C05474=1205.016,78.831,-47.924,-178.902,5.757,148.692
C05475=1205.020,78.581,-47.907,-178.904,5.757,148.692
C05476=1205.025,78.332,-47.889,-178.907,5.756,148.693
C05477=1205.030,78.082,-47.872,-178.910,5.754,148.693
C05478=1205.035,77.833,-47.854,-178.912,5.754,148.694
C05479=1205.039,77.584,-47.836,-178.915,5.753,148.695
C05480=1205.044,77.335,-47.819,-178.917,5.752,148.695
C05481=1205.049,77.085,-47.801,-178.920,5.752,148.696
C05482=1205.055,76.836,-47.784,-178.922,5.750,148.696
C05483=1205.059,76.587,-47.766,-178.925,5.749,148.697
C05484=1205.064,76.337,-47.749,-178.928,5.749,148.698
C05485=1205.069,76.088,-47.731,-178.930,5.748,148.698
C05486=1205.073,75.838,-47.714,-178.933,5.747,148.699
C05487=1205.079,75.590,-47.697,-178.936,5.746,148.699
C05488=1205.084,75.340,-47.680,-178.938,5.745,148.700
C05489=1205.089,75.091,-47.662,-178.940,5.745,148.700
C05490=1205.093,74.841,-47.645,-178.943,5.744,148.701
C05491=1205.099,74.592,-47.628,-178.946,5.742,148.701
C05492=1205.104,74.342,-47.610,-178.948,5.742,148.702
C05493=1205.108,74.093,-47.593,-178.951,5.741,148.703
C05494=1205.113,73.844,-47.575,-178.953,5.740,148.703
C05495=1205.117,73.594,-47.558,-178.956,5.740,148.704
C05496=1205.122,73.345,-47.540,-178.959,5.738,148.704
C05497=1205.128,73.096,-47.523,-178.961,5.737,148.705
C05498=1205.133,72.846,-47.507,-178.964,5.737,148.706
C05499=1205.138,72.597,-47.489,-178.966,5.736,148.706
C05500=1205.143,72.348,-47.472,-178.968,5.735,148.707
C05501=1205.147,72.098,-47.455,-178.972,5.734,148.707
C05502=1205.152,71.849,-47.437,-178.974,5.733,148.708
C05503=1205.157,71.599,-47.420,-178.976,5.732,148.708
C05504=1205.163,71.350,-47.403,-178.979,5.732,148.709
C05505=1205.167,71.101,-47.385,-178.982,5.731,148.710
C05506=1205.172,70.852,-47.369,-178.984,5.730,148.710
C05507=1205.177,70.602,-47.351,-178.987,5.729,148.711
C05508=1205.181,70.353,-47.334,-178.990,5.729,148.711
C05509=1205.187,70.103,-47.317,-178.992,5.728,148.712
C05510=1205.192,69.854,-47.300,-178.994,5.727,148.713
C05511=1205.197,69.605,-47.283,-178.998,5.726,148.713
C05512=1205.201,69.356,-47.266,-179.000,5.725,148.714
C05513=1205.206,69.106,-47.249,-179.002,5.724,148.714
C05514=1205.211,68.856,-47.231,-179.005,5.724,148.715
C05515=1205.216,68.607,-47.215,-179.007,5.723,148.715
C05516=1205.221,68.358,-47.197,-179.010,5.722,148.716
C05517=1205.226,68.109,-47.180,-179.013,5.721,148.717
C05518=1205.231,67.859,-47.163,-179.015,5.720,148.717
C05519=1205.236,67.609,-47.146,-179.018,5.719,148.718
C05520=1205.241,67.360,-47.130,-179.020,5.719,148.718
C05521=1205.246,67.111,-47.112,-179.023,5.718,148.719
C05522=1205.250,66.862,-47.095,-179.026,5.716,148.720
C05523=1205.255,66.612,-47.078,-179.028,5.716,148.720
C05524=1205.260,66.363,-47.062,-179.031,5.715,148.721
C05525=1205.266,66.114,-47.045,-179.033,5.714,148.721
C05526=1205.270,65.864,-47.028,-179.036,5.714,148.722
C05527=1205.275,65.614,-47.011,-179.038,5.713,148.723
C05528=1205.280,65.365,-46.994,-179.041,5.712,148.723
C05529=1205.285,65.116,-46.976,-179.044,5.711,148.724
C05530=1205.290,64.867,-46.960,-179.046,5.711,148.724
C05531=1205.294,64.617,-46.943,-179.049,5.710,148.725
C05532=1205.299,64.368,-46.926,-179.051,5.709,148.726
C05533=1205.305,64.119,-46.910,-179.054,5.709,148.726
C05534=1205.310,63.869,-46.892,-179.056,5.708,148.727
C05535=1205.314,63.620,-46.876,-179.059,5.706,148.727
C05536=1205.319,63.370,-46.859,-179.062,5.706,148.728
C05537=1205.325,63.121,-46.842,-179.064,5.705,148.729
C05538=1205.329,62.871,-46.825,-179.067,5.704,148.729
C05539=1205.334,62.622,-46.808,-179.069,5.704,148.730
C05540=1205.339,62.373,-46.792,-179.072,5.703,148.730
C05541=1205.344,62.123,-46.775,-179.074,5.702,148.731
C05542=1205.349,61.874,-46.758,-179.077,5.701,148.731
C05543=1205.354,61.625,-46.742,-179.080,5.700,148.732
C05544=1205.359,61.375,-46.725,-179.082,5.700,148.733
C05545=1205.364,61.126,-46.708,-179.085,5.699,148.733
C05546=1205.368,60.876,-46.691,-179.087,5.698,148.734
C05547=1205.373,60.627,-46.675,-179.090,5.698,148.735
C05548=1205.379,60.377,-46.657,-179.092,5.697,148.735
C05549=1205.383,60.128,-46.641,-179.095,5.695,148.736
C05550=1205.388,59.879,-46.624,-179.098,5.695,148.736
C05551=1205.393,59.629,-46.607,-179.100,5.694,148.737
C05552=1205.398,59.380,-46.590,-179.103,5.693,148.737
C05553=1205.403,59.131,-46.575,-179.105,5.693,148.738
C05554=1205.408,58.881,-46.558,-179.108,5.692,148.739
C05555=1205.414,58.632,-46.541,-179.110,5.691,148.739
C05556=1205.418,58.382,-46.525,-179.113,5.691,148.740
C05557=1205.422,58.133,-46.508,-179.116,5.690,148.741
C05558=1205.428,57.884,-46.492,-179.118,5.689,148.741
C05559=1205.433,57.634,-46.474,-179.121,5.688,148.742
C05560=1205.438,57.384,-46.458,-179.123,5.688,148.742
C05561=1205.443,57.136,-46.442,-179.126,5.687,148.743
C05562=1205.447,56.886,-46.425,-179.128,5.686,148.743
C05563=1205.453,56.637,-46.409,-179.131,5.686,148.744
C05564=1205.457,56.387,-46.392,-179.133,5.685,148.745
C05565=1205.462,56.137,-46.376,-179.137,5.684,148.745
C05566=1205.467,55.889,-46.360,-179.139,5.683,148.746
C05567=1205.473,55.639,-46.342,-179.141,5.682,148.746
C05568=1205.478,55.371,-46.325,-179.144,5.682,148.747
C05569=1205.483,55.102,-46.307,-179.147,5.681,148.748
C05570=1205.488,54.834,-46.290,-179.150,5.680,148.748
C05571=1205.494,54.565,-46.272,-179.152,5.679,148.749
C05572=1205.499,54.316,-46.255,-179.155,5.679,148.750
C05573=1205.503,54.066,-46.239,-179.157,5.678,148.750
C05574=1205.509,53.817,-46.223,-179.160,5.677,148.751
C05575=1205.513,53.567,-46.206,-179.162,5.677,148.752
C05576=1205.518,53.318,-46.190,-179.165,5.676,148.752
C05577=1205.523,53.068,-46.174,-179.167,5.675,148.753
C05578=1205.529,52.819,-46.157,-179.170,5.674,148.753
C05579=1205.533,52.570,-46.141,-179.173,5.673,148.754
C05580=1205.539,52.320,-46.125,-179.175,5.672,148.754
C05581=1205.543,52.071,-46.108,-179.178,5.672,148.755
C05582=1205.548,51.821,-46.092,-179.181,5.671,148.756
C05583=1205.553,51.572,-46.076,-179.183,5.671,148.756
C05584=1205.557,51.323,-46.059,-179.185,5.670,148.757
C05585=1205.563,51.073,-46.044,-179.188,5.669,148.758
C05586=1205.567,50.824,-46.027,-179.191,5.669,148.758
C05587=1205.572,50.575,-46.011,-179.193,5.668,148.759
C05588=1205.577,50.325,-45.995,-179.195,5.667,148.759
C05589=1205.583,50.076,-45.978,-179.198,5.667,148.760
C05590=1205.588,49.826,-45.962,-179.201,5.665,148.761
C05591=1205.593,49.577,-45.946,-179.204,5.665,148.761
C05592=1205.597,49.327,-45.929,-179.206,5.664,148.762
C05593=1205.603,49.078,-45.913,-179.209,5.663,148.762
C05594=1205.607,48.828,-45.897,-179.211,5.663,148.763
C05595=1205.613,48.579,-45.881,-179.214,5.662,148.764
C05596=1205.617,48.329,-45.864,-179.216,5.661,148.764
C05597=1205.622,48.080,-45.849,-179.219,5.661,148.765
C05598=1205.627,47.831,-45.832,-179.221,5.660,148.766
C05599=1205.632,47.581,-45.817,-179.224,5.660,148.766
C05600=1205.637,47.332,-45.800,-179.226,5.659,148.767
C05601=1205.642,47.082,-45.784,-179.229,5.658,148.767
C05602=1205.647,46.834,-45.768,-179.231,5.658,148.768
C05603=1205.652,46.583,-45.752,-179.234,5.657,148.769
C05604=1205.657,46.334,-45.737,-179.237,5.656,148.769
C05605=1205.662,46.085,-45.720,-179.239,5.655,148.770
C05606=1205.667,45.835,-45.704,-179.242,5.654,148.770
C05607=1205.672,45.586,-45.688,-179.245,5.654,148.771
C05608=1205.677,45.336,-45.672,-179.247,5.653,148.772
C05609=1205.682,45.087,-45.655,-179.249,5.653,148.772
C05610=1205.686,44.838,-45.640,-179.252,5.652,148.773
C05611=1205.692,44.588,-45.625,-179.255,5.651,148.774
C05612=1205.696,44.339,-45.608,-179.257,5.651,148.774
C05613=1205.702,44.089,-45.593,-179.260,5.650,148.775
C05614=1205.706,43.839,-45.577,-179.262,5.649,148.775
C05615=1205.711,43.591,-45.560,-179.265,5.649,148.776
C05616=1205.717,43.341,-45.545,-179.267,5.648,148.777
C05617=1205.722,43.091,-45.529,-179.270,5.648,148.777
C05618=1205.727,42.842,-45.512,-179.272,5.647,148.778
C05619=1205.731,42.592,-45.496,-179.275,5.646,148.779
C05620=1205.737,42.343,-45.481,-179.278,5.646,148.779
C05621=1205.741,42.094,-45.465,-179.280,5.645,148.780
C05622=1205.746,41.844,-45.449,-179.282,5.644,148.780
C05623=1205.751,41.595,-45.434,-179.285,5.644,148.781
C05624=1205.756,41.345,-45.418,-179.288,5.643,148.782
C05625=1205.761,41.096,-45.401,-179.291,5.642,148.782
C05626=1205.767,40.846,-45.386,-179.293,5.641,148.783
C05627=1205.771,40.596,-45.370,-179.296,5.641,148.783
C05628=1205.776,40.347,-45.355,-179.298,5.640,148.784
C05629=1205.781,40.098,-45.339,-179.301,5.640,148.785
C05630=1205.786,39.848,-45.323,-179.304,5.639,148.785
C05631=1205.791,39.599,-45.307,-179.306,5.638,148.786
C05632=1205.797,39.350,-45.291,-179.308,5.638,148.787
C05633=1205.800,39.100,-45.275,-179.311,5.637,148.787
C05634=1205.806,38.851,-45.260,-179.314,5.637,148.788
C05635=1205.811,38.602,-45.244,-179.316,5.636,148.788
C05636=1205.816,38.351,-45.228,-179.318,5.635,148.789
C05637=1205.821,38.102,-45.213,-179.321,5.635,148.790
C05638=1205.826,37.853,-45.198,-179.324,5.634,148.790
C05639=1205.831,37.604,-45.181,-179.326,5.634,148.791
C05640=1205.836,37.354,-45.165,-179.328,5.633,148.792
C05641=1205.841,37.105,-45.150,-179.331,5.632,148.792
C05642=1205.845,36.855,-45.134,-179.334,5.632,148.793
C05643=1205.851,36.606,-45.119,-179.336,5.631,148.794
C05644=1205.856,36.356,-45.103,-179.339,5.630,148.794
C05645=1205.862,36.107,-45.088,-179.341,5.630,148.795
C05646=1205.866,35.857,-45.072,-179.344,5.629,148.795
C05647=1205.871,35.608,-45.057,-179.347,5.629,148.796
C05648=1205.876,35.358,-45.041,-179.349,5.628,148.797
C05649=1205.881,35.109,-45.024,-179.352,5.627,148.797
C05650=1205.885,34.860,-45.009,-179.354,5.627,148.798
C05651=1205.891,34.610,-44.994,-179.357,5.626,148.799
C05652=1205.896,34.361,-44.978,-179.359,5.626,148.799
C05653=1205.900,34.111,-44.963,-179.362,5.625,148.800
C05654=1205.906,33.862,-44.947,-179.365,5.624,148.801
C05655=1205.911,33.612,-44.932,-179.367,5.624,148.801
C05656=1205.916,33.363,-44.917,-179.369,5.623,148.802
C05657=1205.921,33.113,-44.901,-179.372,5.623,148.802
C05658=1205.926,32.864,-44.885,-179.375,5.622,148.803
C05659=1205.931,32.614,-44.870,-179.377,5.621,148.804
C05660=1205.936,32.365,-44.855,-179.379,5.621,148.804
C05661=1205.941,32.115,-44.839,-179.382,5.620,148.805
C05662=1205.945,31.866,-44.824,-179.385,5.620,148.805
C05663=1205.951,31.616,-44.808,-179.387,5.619,148.806
C05664=1205.956,31.367,-44.794,-179.390,5.618,148.807
C05665=1205.961,31.117,-44.778,-179.392,5.618,148.807
C05666=1205.966,30.867,-44.762,-179.395,5.617,148.808
C05667=1205.971,30.618,-44.747,-179.397,5.617,148.809
C05668=1205.976,30.369,-44.732,-179.400,5.616,148.809
C05669=1205.981,30.120,-44.717,-179.403,5.615,148.810
C05670=1205.986,29.870,-44.701,-179.405,5.615,148.810
C05671=1205.991,29.620,-44.685,-179.407,5.614,148.811
C05672=1205.996,29.351,-44.669,-179.410,5.614,148.812
C05673=1206.001,29.083,-44.652,-179.413,5.613,148.812
C05674=1206.007,28.814,-44.637,-179.415,5.613,148.813
C05675=1206.012,28.546,-44.620,-179.418,5.612,148.814
C05676=1206.017,28.296,-44.604,-179.421,5.611,148.815
C05677=1206.022,28.046,-44.590,-179.423,5.611,148.815
C05678=1206.028,27.797,-44.574,-179.426,5.610,148.816
C05679=1206.032,27.548,-44.559,-179.429,5.610,148.817
C05680=1206.037,27.298,-44.543,-179.431,5.609,148.817
C05681=1206.042,27.049,-44.528,-179.433,5.608,148.818
C05682=1206.048,26.799,-44.513,-179.436,5.608,148.818
C05683=1206.052,26.550,-44.498,-179.439,5.607,148.819
C05684=1206.058,26.300,-44.483,-179.441,5.607,148.820
C05685=1206.062,26.051,-44.468,-179.444,5.606,148.820
C05686=1206.068,25.802,-44.452,-179.446,5.606,148.821
C05687=1206.072,25.551,-44.438,-179.449,5.605,148.822
C05688=1206.077,25.302,-44.422,-179.451,5.604,148.822
C05689=1206.082,25.053,-44.407,-179.454,5.604,148.823
C05690=1206.088,24.803,-44.392,-179.457,5.603,148.824
C05691=1206.092,24.554,-44.377,-179.459,5.603,148.824
C05692=1206.098,24.304,-44.362,-179.462,5.602,148.825
C05693=1206.102,24.055,-44.347,-179.464,5.601,148.825
C05694=1206.107,23.806,-44.332,-179.467,5.601,148.826
C05695=1206.112,23.555,-44.316,-179.469,5.601,148.827
C05696=1206.117,23.306,-44.301,-179.471,5.600,148.827
C05697=1206.123,23.056,-44.287,-179.474,5.600,148.828
C05698=1206.127,22.807,-44.272,-179.476,5.599,148.829
C05699=1206.133,22.557,-44.257,-179.479,5.599,148.829
C05700=1206.138,22.308,-44.242,-179.482,5.598,148.830
C05701=1206.142,22.059,-44.227,-179.484,5.598,148.831
C05702=1206.148,21.809,-44.212,-179.486,5.597,148.831
C05703=1206.153,21.560,-44.197,-179.489,5.596,148.832
C05704=1206.158,21.311,-44.181,-179.492,5.596,148.832
C05705=1206.163,21.061,-44.167,-179.494,5.595,148.833
C05706=1206.167,20.812,-44.152,-179.497,5.595,148.834
C05707=1206.173,20.562,-44.137,-179.500,5.594,148.834
C05708=1206.178,20.313,-44.122,-179.502,5.593,148.835
C05709=1206.183,20.063,-44.108,-179.505,5.593,148.836
C05710=1206.188,19.814,-44.092,-179.507,5.592,148.836
C05711=1206.192,19.564,-44.077,-179.509,5.593,148.837
C05712=1206.197,19.314,-44.063,-179.512,5.592,148.838
C05713=1206.203,19.065,-44.047,-179.515,5.592,148.838
C05714=1206.208,18.815,-44.033,-179.517,5.591,148.839
C05715=1206.212,18.566,-44.018,-179.519,5.590,148.839
C05716=1206.218,18.316,-44.003,-179.522,5.590,148.840
C05717=1206.223,18.067,-43.988,-179.525,5.589,148.841
C05718=1206.227,17.817,-43.974,-179.527,5.589,148.841
C05719=1206.233,17.568,-43.958,-179.530,5.588,148.842
C05720=1206.238,17.318,-43.944,-179.532,5.587,148.843
C05721=1206.242,17.069,-43.929,-179.535,5.587,148.843
C05722=1206.247,16.819,-43.914,-179.537,5.586,148.844
C05723=1206.253,16.569,-43.900,-179.540,5.586,148.845
C05724=1206.258,16.320,-43.885,-179.542,5.586,148.845
C05725=1206.263,16.070,-43.870,-179.545,5.586,148.846
C05726=1206.267,15.821,-43.855,-179.547,5.585,148.846
C05727=1206.273,15.571,-43.840,-179.550,5.584,148.847
C05728=1206.278,15.322,-43.825,-179.552,5.584,148.848
C05729=1206.283,15.072,-43.811,-179.555,5.583,148.849
C05730=1206.288,14.823,-43.797,-179.558,5.583,148.849
C05731=1206.294,14.574,-43.782,-179.560,5.582,148.850
C05732=1206.299,14.324,-43.767,-179.563,5.582,148.851
C05733=1206.304,14.074,-43.753,-179.565,5.581,148.851
C05734=1206.308,13.825,-43.738,-179.568,5.580,148.852
C05735=1206.314,13.575,-43.723,-179.570,5.581,148.852
C05736=1206.319,13.326,-43.709,-179.572,5.580,148.853
C05737=1206.323,13.077,-43.694,-179.575,5.580,148.854
C05738=1206.328,12.827,-43.680,-179.578,5.579,148.854
C05739=1206.333,12.577,-43.665,-179.580,5.578,148.855
C05740=1206.338,12.328,-43.650,-179.582,5.578,148.856
C05741=1206.344,12.078,-43.636,-179.585,5.577,148.856
C05742=1206.349,11.828,-43.621,-179.588,5.577,148.857
C05743=1206.353,11.579,-43.606,-179.590,5.576,148.858
C05744=1206.358,11.330,-43.592,-179.593,5.576,148.858
C05745=1206.364,11.081,-43.578,-179.595,5.576,148.859
C05746=1206.369,10.831,-43.564,-179.597,5.575,148.859
C05747=1206.374,10.581,-43.548,-179.600,5.574,148.860
C05748=1206.379,10.332,-43.534,-179.603,5.574,148.861
C05749=1206.384,10.082,-43.520,-179.605,5.573,148.862
C05750=1206.389,9.832,-43.505,-179.608,5.573,148.862
C05751=1206.394,9.583,-43.490,-179.611,5.572,148.863
C05752=1206.399,9.333,-43.476,-179.613,5.572,148.864
C05753=1206.404,9.084,-43.462,-179.615,5.572,148.864
C05754=1206.409,8.835,-43.448,-179.617,5.571,148.865
C05755=1206.414,8.585,-43.434,-179.620,5.571,148.865
C05756=1206.419,8.336,-43.418,-179.623,5.570,148.866
C05757=1206.424,8.086,-43.404,-179.625,5.570,148.867
C05758=1206.429,7.836,-43.390,-179.628,5.569,148.867
C05759=1206.434,7.587,-43.375,-179.630,5.568,148.868
C05760=1206.439,7.337,-43.361,-179.633,5.568,148.869
C05761=1206.444,7.087,-43.347,-179.635,5.567,148.869
C05762=1206.450,6.838,-43.333,-179.638,5.568,148.870
C05763=1206.454,6.589,-43.318,-179.640,5.567,148.871
C05764=1206.459,6.339,-43.304,-179.643,5.567,148.871
C05765=1206.464,6.090,-43.289,-179.646,5.566,148.872
C05766=1206.469,5.840,-43.275,-179.648,5.565,148.873
C05767=1206.474,5.590,-43.261,-179.650,5.565,148.873
C05768=1206.480,5.341,-43.247,-179.653,5.564,148.874
C05769=1206.485,5.091,-43.232,-179.655,5.565,148.875
C05770=1206.490,4.842,-43.218,-179.658,5.564,148.875
C05771=1206.495,4.592,-43.204,-179.660,5.564,148.876
C05772=1206.500,4.342,-43.190,-179.663,5.563,148.877
C05773=1206.505,4.093,-43.176,-179.666,5.563,148.877
C05774=1206.510,3.844,-43.161,-179.668,5.562,148.878
C05775=1206.515,3.594,-43.147,-179.670,5.561,148.878
C05776=1206.520,3.325,-43.131,-179.673,5.561,148.879
C05777=1206.526,3.056,-43.116,-179.676,5.560,148.880
C05778=1206.531,2.787,-43.101,-179.679,5.560,148.881
C05779=1206.537,2.518,-43.086,-179.682,5.560,148.881
C05780=1206.542,2.268,-43.072,-179.683,5.560,148.882
C05781=1206.547,2.019,-43.058,-179.686,5.559,148.883
C05782=1206.552,1.769,-43.043,-179.688,5.559,148.883
C05783=1206.557,1.520,-43.029,-179.691,5.558,148.884
C05784=1206.562,1.270,-43.015,-179.694,5.558,148.885
C05785=1206.567,1.021,-43.001,-179.696,5.557,148.885
C05786=1206.572,0.771,-42.987,-179.699,5.557,148.886
C05787=1206.578,0.522,-42.973,-179.701,5.557,148.887
C05788=1206.583,0.272,-42.958,-179.703,5.556,148.887
C05789=1206.588,0.022,-42.944,-179.706,5.556,148.888
C05790=1206.592,-0.228,-42.931,-179.709,5.555,148.889
C05791=1206.598,-0.477,-42.917,-179.711,5.555,148.889
C05792=1206.603,-0.726,-42.903,-179.714,5.554,148.890
C05793=1206.608,-0.976,-42.889,-179.716,5.554,148.891
C05794=1206.613,-1.226,-42.874,-179.719,5.554,148.891
C05795=1206.618,-1.475,-42.860,-179.721,5.553,148.892
C05796=1206.623,-1.724,-42.846,-179.723,5.552,148.892
C05797=1206.627,-1.974,-42.833,-179.726,5.552,148.893
C05798=1206.633,-2.223,-42.819,-179.729,5.551,148.894
C05799=1206.638,-2.473,-42.805,-179.731,5.552,148.895
C05800=1206.643,-2.723,-42.791,-179.734,5.551,148.895
C05801=1206.648,-2.973,-42.777,-179.736,5.551,148.896
C05802=1206.654,-3.222,-42.763,-179.739,5.550,148.897
C05803=1206.658,-3.472,-42.750,-179.741,5.549,148.897
C05804=1206.663,-3.721,-42.735,-179.744,5.549,148.898
C05805=1206.669,-3.970,-42.721,-179.746,5.549,148.898
C05806=1206.674,-4.220,-42.707,-179.748,5.549,148.899
C05807=1206.678,-4.470,-42.693,-179.751,5.548,148.900
C05808=1206.684,-4.719,-42.680,-179.754,5.548,148.901
C05809=1206.689,-4.969,-42.666,-179.756,5.547,148.901
C05810=1206.694,-5.219,-42.652,-179.759,5.547,148.902
C05811=1206.699,-5.468,-42.638,-179.761,5.547,148.902
C05812=1206.704,-5.718,-42.624,-179.763,5.546,148.903
C05813=1206.709,-5.967,-42.611,-179.766,5.546,148.904
C05814=1206.714,-6.216,-42.597,-179.769,5.545,148.904
C05815=1206.719,-6.467,-42.583,-179.771,5.545,148.905
C05816=1206.724,-6.716,-42.569,-179.773,5.545,148.906
C05817=1206.729,-6.965,-42.556,-179.776,5.545,148.906
C05818=1206.734,-7.215,-42.541,-179.779,5.544,148.907
C05819=1206.739,-7.465,-42.528,-179.781,5.543,148.908
C05820=1206.744,-7.714,-42.514,-179.783,5.543,148.908
C05821=1206.749,-7.963,-42.500,-179.785,5.543,148.909
C05822=1206.755,-8.213,-42.487,-179.788,5.543,148.910
C05823=1206.760,-8.463,-42.473,-179.791,5.542,148.910
C05824=1206.764,-8.713,-42.460,-179.793,5.542,148.911
C05825=1206.770,-8.962,-42.446,-179.796,5.541,148.912
C05826=1206.775,-9.212,-42.431,-179.798,5.541,148.912
C05827=1206.780,-9.461,-42.419,-179.800,5.541,148.913
C05828=1206.785,-9.711,-42.405,-179.803,5.540,148.914
C05829=1206.790,-9.960,-42.390,-179.806,5.540,148.914
C05830=1206.795,-10.210,-42.378,-179.808,5.539,148.915
C05831=1206.800,-10.459,-42.363,-179.810,5.539,148.916
C05832=1206.806,-10.709,-42.350,-179.813,5.539,148.916
C05833=1206.810,-10.958,-42.337,-179.816,5.538,148.917
C05834=1206.815,-11.209,-42.323,-179.818,5.538,148.918
C05835=1206.821,-11.458,-42.309,-179.821,5.537,148.918
C05836=1206.826,-11.708,-42.296,-179.823,5.537,148.919
C05837=1206.831,-11.957,-42.282,-179.825,5.537,148.920
C05838=1206.835,-12.206,-42.269,-179.828,5.536,148.920
C05839=1206.841,-12.456,-42.255,-179.831,5.536,148.921
C05840=1206.846,-12.705,-42.241,-179.833,5.535,148.922
C05841=1206.851,-12.955,-42.228,-179.835,5.536,148.922
C05842=1206.856,-13.204,-42.214,-179.838,5.535,148.923
C05843=1206.861,-13.455,-42.201,-179.840,5.534,148.924
C05844=1206.866,-13.703,-42.187,-179.843,5.534,148.924
C05845=1206.872,-13.954,-42.174,-179.845,5.533,148.925
C05846=1206.877,-14.203,-42.161,-179.848,5.534,148.926
C05847=1206.882,-14.453,-42.147,-179.850,5.533,148.926
C05848=1206.887,-14.702,-42.134,-179.853,5.533,148.927
C05849=1206.892,-14.952,-42.120,-179.855,5.532,148.928
C05850=1206.898,-15.201,-42.107,-179.858,5.533,148.928
C05851=1206.902,-15.451,-42.093,-179.860,5.532,148.929
C05852=1206.908,-15.701,-42.080,-179.862,5.531,148.930
C05853=1206.912,-15.951,-42.067,-179.865,5.531,148.930
C05854=1206.918,-16.200,-42.053,-179.868,5.530,148.931
C05855=1206.922,-16.450,-42.040,-179.870,5.531,148.932
C05856=1206.928,-16.699,-42.026,-179.872,5.530,148.932
C05857=1206.932,-16.949,-42.013,-179.875,5.530,148.933
C05858=1206.938,-17.198,-42.000,-179.878,5.529,148.934
C05859=1206.942,-17.448,-41.986,-179.880,5.529,148.934
C05860=1206.948,-17.697,-41.973,-179.882,5.529,148.935
C05861=1206.953,-17.947,-41.960,-179.885,5.528,148.936
C05862=1206.958,-18.196,-41.946,-179.887,5.528,148.936
C05863=1206.963,-18.446,-41.933,-179.889,5.528,148.937
C05864=1206.969,-18.696,-41.920,-179.892,5.527,148.938
C05865=1206.973,-18.945,-41.906,-179.895,5.527,148.938
C05866=1206.979,-19.195,-41.893,-179.897,5.526,148.939
C05867=1206.983,-19.445,-41.880,-179.900,5.526,148.940
C05868=1206.989,-19.694,-41.866,-179.902,5.526,148.940
C05869=1206.994,-19.943,-41.854,-179.904,5.525,148.941
C05870=1206.999,-20.194,-41.840,-179.907,5.525,148.942
C05871=1207.004,-20.443,-41.828,-179.910,5.524,148.942
C05872=1207.009,-20.692,-41.814,-179.912,5.525,148.943
C05873=1207.014,-20.942,-41.801,-179.914,5.524,148.944
C05874=1207.019,-21.192,-41.788,-179.917,5.524,148.944
C05875=1207.025,-21.442,-41.774,-179.920,5.523,148.945
C05876=1207.030,-21.690,-41.761,-179.922,5.524,148.946
C05877=1207.035,-21.941,-41.748,-179.924,5.523,148.946
C05878=1207.040,-22.190,-41.735,-179.927,5.522,148.947
C05879=1207.045,-22.440,-41.722,-179.929,5.522,148.948
C05880=1207.051,-22.709,-41.707,-179.931,5.522,148.948
C05881=1207.056,-22.979,-41.693,-179.934,5.522,148.949
C05882=1207.061,-23.248,-41.679,-179.937,5.522,148.950
C05883=1207.067,-23.517,-41.665,-179.940,5.521,148.951
C05884=1207.072,-23.767,-41.652,-179.942,5.521,148.951
C05885=1207.077,-24.017,-41.639,-179.945,5.520,148.952
C05886=1207.082,-24.267,-41.626,-179.947,5.520,148.953
C05887=1207.087,-24.516,-41.613,-179.949,5.520,148.953
C05888=1207.093,-24.766,-41.600,-179.952,5.519,148.954
C05889=1207.097,-25.015,-41.586,-179.955,5.519,148.955
C05890=1207.103,-25.265,-41.574,-179.957,5.519,148.955
C05891=1207.107,-25.515,-41.561,-179.959,5.519,148.956
C05892=1207.113,-25.764,-41.547,-179.962,5.518,148.957
C05893=1207.118,-26.013,-41.535,-179.965,5.518,148.957
C05894=1207.123,-26.263,-41.522,-179.967,5.518,148.958
C05895=1207.128,-26.513,-41.509,-179.969,5.517,148.959
C05896=1207.134,-26.762,-41.496,-179.972,5.517,148.959
C05897=1207.138,-27.012,-41.483,-179.974,5.517,148.960
C05898=1207.144,-27.262,-41.470,-179.976,5.516,148.961
C05899=1207.149,-27.511,-41.457,-179.979,5.516,148.961
C05900=1207.153,-27.761,-41.444,-179.982,5.515,148.962
C05901=1207.158,-28.010,-41.431,-179.984,5.516,148.963
C05902=1207.164,-28.260,-41.418,-179.986,5.515,148.963
C05903=1207.169,-28.510,-41.405,-179.989,5.515,148.964
C05904=1207.174,-28.759,-41.392,-179.991,5.514,148.965
C05905=1207.180,-29.009,-41.379,-179.993,5.514,148.965
C05906=1207.184,-29.259,-41.366,-179.996,5.514,148.966
C05907=1207.189,-29.508,-41.354,-179.999,5.513,148.967
C05908=1207.195,-29.757,-41.341,179.999,5.514,148.967
C05909=1207.199,-30.007,-41.328,179.997,5.513,148.968
C05910=1207.205,-30.257,-41.315,179.994,5.513,148.969
C05911=1207.210,-30.506,-41.302,179.991,5.512,148.969
C05912=1207.215,-30.757,-41.290,179.989,5.513,148.970
C05913=1207.220,-31.006,-41.277,179.987,5.512,148.971
C05914=1207.226,-31.256,-41.264,179.984,5.511,148.971
C05915=1207.231,-31.505,-41.252,179.982,5.511,148.972
C05916=1207.236,-31.755,-41.239,179.980,5.511,148.973
C05917=1207.241,-32.005,-41.226,179.977,5.511,148.973
C05918=1207.246,-32.254,-41.213,179.974,5.510,148.974
C05919=1207.251,-32.504,-41.200,179.972,5.511,148.975
C05920=1207.256,-32.754,-41.187,179.970,5.510,148.976
C05921=1207.261,-33.003,-41.175,179.967,5.510,148.976
C05922=1207.266,-33.252,-41.162,179.965,5.510,148.977
C05923=1207.271,-33.502,-41.149,179.963,5.509,148.977
C05924=1207.276,-33.752,-41.137,179.960,5.509,148.978
C05925=1207.282,-34.002,-41.124,179.957,5.508,148.979
C05926=1207.287,-34.251,-41.111,179.955,5.508,148.980
C05927=1207.292,-34.501,-41.098,179.953,5.508,148.980
C05928=1207.297,-34.750,-41.086,179.950,5.508,148.981
C05929=1207.302,-35.000,-41.073,179.948,5.508,148.982
C05930=1207.308,-35.250,-41.061,179.945,5.507,148.982
C05931=1207.313,-35.499,-41.049,179.943,5.507,148.983
C05932=1207.317,-35.749,-41.036,179.940,5.506,148.983
C05933=1207.323,-35.999,-41.023,179.938,5.506,148.984
C05934=1207.328,-36.248,-41.010,179.936,5.506,148.985
C05935=1207.334,-36.498,-40.998,179.933,5.506,148.986
C05936=1207.339,-36.747,-40.985,179.931,5.506,148.986
C05937=1207.343,-36.997,-40.972,179.928,5.505,148.987
C05938=1207.348,-37.247,-40.960,179.926,5.505,148.988
C05939=1207.354,-37.496,-40.948,179.924,5.505,148.988
C05940=1207.359,-37.746,-40.935,179.921,5.504,148.989
C05941=1207.364,-37.995,-40.923,179.919,5.504,148.990
C05942=1207.369,-38.245,-40.910,179.917,5.504,148.990
C05943=1207.374,-38.495,-40.898,179.914,5.504,148.991
C05944=1207.379,-38.744,-40.885,179.911,5.503,148.992
C05945=1207.384,-38.994,-40.873,179.909,5.503,148.992
C05946=1207.390,-39.244,-40.860,179.906,5.503,148.993
C05947=1207.396,-39.493,-40.848,179.904,5.503,148.994
C05948=1207.400,-39.743,-40.835,179.902,5.502,148.994
C05949=1207.405,-39.993,-40.822,179.900,5.502,148.995
C05950=1207.411,-40.243,-40.810,179.897,5.502,148.996
C05951=1207.416,-40.492,-40.798,179.894,5.501,148.996
C05952=1207.421,-40.741,-40.785,179.892,5.502,148.997
C05953=1207.426,-40.991,-40.773,179.889,5.501,148.998
C05954=1207.431,-41.241,-40.760,179.887,5.501,148.998
C05955=1207.436,-41.491,-40.748,179.885,5.501,148.999
C05956=1207.441,-41.740,-40.736,179.882,5.501,149.000
C05957=1207.447,-41.990,-40.723,179.880,5.500,149.000
C05958=1207.452,-42.240,-40.711,179.878,5.500,149.001
C05959=1207.456,-42.489,-40.699,179.875,5.500,149.002
C05960=1207.461,-42.738,-40.687,179.872,5.499,149.002
C05961=1207.466,-42.989,-40.674,179.870,5.499,149.003
C05962=1207.471,-43.238,-40.662,179.868,5.499,149.004
C05963=1207.477,-43.488,-40.650,179.865,5.499,149.004
C05964=1207.482,-43.737,-40.637,179.863,5.499,149.005
C05965=1207.487,-43.987,-40.625,179.860,5.498,149.006
C05966=1207.493,-44.236,-40.613,179.858,5.498,149.006
C05967=1207.498,-44.486,-40.601,179.856,5.498,149.007
C05968=1207.503,-44.736,-40.588,179.853,5.497,149.008
C05969=1207.508,-44.985,-40.576,179.851,5.497,149.008
C05970=1207.514,-45.235,-40.564,179.849,5.497,149.009
C05971=1207.518,-45.485,-40.551,179.846,5.497,149.010
C05972=1207.524,-45.735,-40.539,179.843,5.496,149.011
C05973=1207.528,-45.984,-40.527,179.841,5.497,149.011
C05974=1207.533,-46.234,-40.515,179.839,5.496,149.012
C05975=1207.539,-46.483,-40.502,179.836,5.495,149.012
C05976=1207.544,-46.733,-40.491,179.834,5.496,149.013
C05977=1207.549,-46.982,-40.478,179.832,5.495,149.014
C05978=1207.555,-47.232,-40.466,179.829,5.495,149.015
C05979=1207.560,-47.482,-40.454,179.827,5.495,149.015
C05980=1207.565,-47.732,-40.442,179.824,5.495,149.016
C05981=1207.570,-47.981,-40.430,179.822,5.494,149.017
C05982=1207.575,-48.231,-40.418,179.819,5.495,149.017
C05983=1207.580,-48.480,-40.406,179.817,5.494,149.018
C05984=1207.586,-48.751,-40.393,179.815,5.493,149.019
C05985=1207.591,-49.021,-40.379,179.811,5.493,149.019
C05986=1207.597,-49.291,-40.366,179.809,5.494,149.020
C05987=1207.603,-49.561,-40.353,179.807,5.493,149.021
C05988=1207.608,-49.811,-40.341,179.804,5.493,149.022
C05989=1207.612,-50.060,-40.329,179.801,5.492,149.022
C05990=1207.618,-50.310,-40.317,179.800,5.492,149.023
C05991=1207.623,-50.559,-40.305,179.797,5.492,149.023
C05992=1207.628,-50.809,-40.293,179.795,5.492,149.024
C05993=1207.634,-51.059,-40.281,179.792,5.492,149.025
C05994=1207.638,-51.308,-40.269,179.790,5.491,149.026
C05995=1207.644,-51.558,-40.257,179.788,5.492,149.026
C05996=1207.649,-51.808,-40.245,179.785,5.491,149.027
C05997=1207.654,-52.057,-40.232,179.782,5.491,149.028
C05998=1207.659,-52.307,-40.221,179.780,5.491,149.028
C05999=1207.664,-52.557,-40.209,179.778,5.490,149.029
C06000=1207.669,-52.806,-40.197,179.775,5.490,149.030
C06001=1207.675,-53.056,-40.185,179.773,5.490,149.030
C06002=1207.680,-53.306,-40.174,179.771,5.490,149.031
C06003=1207.685,-53.556,-40.162,179.768,5.489,149.032
C06004=1207.690,-53.805,-40.149,179.766,5.489,149.032
C06005=1207.696,-54.055,-40.137,179.763,5.489,149.033
C06006=1207.700,-54.304,-40.126,179.761,5.489,149.034
C06007=1207.706,-54.554,-40.114,179.759,5.489,149.034
C06008=1207.711,-54.804,-40.101,179.756,5.488,149.035
C06009=1207.715,-55.053,-40.090,179.754,5.488,149.036
C06010=1207.721,-55.303,-40.078,179.752,5.488,149.036
C06011=1207.726,-55.553,-40.066,179.749,5.488,149.037
C06012=1207.731,-55.801,-40.055,179.747,5.488,149.038
C06013=1207.737,-56.051,-40.043,179.744,5.487,149.038
C06014=1207.742,-56.301,-40.031,179.742,5.487,149.039
C06015=1207.747,-56.551,-40.020,179.740,5.487,149.040
C06016=1207.752,-56.801,-40.008,179.737,5.486,149.040
C06017=1207.757,-57.050,-39.995,179.735,5.487,149.041
C06018=1207.762,-57.300,-39.984,179.732,5.486,149.042
C06019=1207.768,-57.550,-39.972,179.730,5.486,149.042
C06020=1207.773,-57.800,-39.960,179.728,5.486,149.043
C06021=1207.778,-58.049,-39.949,179.725,5.486,149.044
C06022=1207.783,-58.299,-39.937,179.723,5.485,149.044
C06023=1207.788,-58.549,-39.924,179.721,5.485,149.045
C06024=1207.793,-58.798,-39.913,179.718,5.485,149.046
C06025=1207.799,-59.047,-39.901,179.716,5.485,149.046
C06026=1207.804,-59.297,-39.890,179.713,5.485,149.047
C06027=1207.809,-59.547,-39.878,179.711,5.484,149.048
C06028=1207.814,-59.797,-39.866,179.709,5.485,149.049
C06029=1207.819,-60.047,-39.855,179.706,5.484,149.049
C06030=1207.825,-60.297,-39.843,179.704,5.484,149.050
C06031=1207.829,-60.546,-39.832,179.702,5.484,149.050
C06032=1207.835,-60.796,-39.820,179.699,5.483,149.051
C06033=1207.840,-61.046,-39.808,179.697,5.484,149.052
C06034=1207.845,-61.294,-39.797,179.694,5.483,149.053
C06035=1207.851,-61.544,-39.785,179.692,5.483,149.053
C06036=1207.855,-61.794,-39.773,179.689,5.483,149.054
C06037=1207.861,-62.044,-39.761,179.687,5.482,149.054
C06038=1207.865,-62.293,-39.750,179.685,5.483,149.055
C06039=1207.871,-62.543,-39.738,179.683,5.482,149.056
C06040=1207.876,-62.793,-39.727,179.680,5.482,149.057
C06041=1207.882,-63.042,-39.715,179.678,5.482,149.057
C06042=1207.887,-63.292,-39.704,179.675,5.482,149.058
C06043=1207.892,-63.542,-39.692,179.673,5.482,149.059
C06044=1207.897,-63.792,-39.680,179.670,5.482,149.059
C06045=1207.902,-64.041,-39.669,179.668,5.481,149.060
C06046=1207.907,-64.291,-39.657,179.666,5.481,149.061
C06047=1207.913,-64.540,-39.646,179.663,5.481,149.061
C06048=1207.918,-64.790,-39.634,179.661,5.481,149.062
C06049=1207.923,-65.040,-39.623,179.659,5.481,149.063
C06050=1207.928,-65.290,-39.612,179.656,5.480,149.063
C06051=1207.933,-65.540,-39.601,179.654,5.480,149.064
C06052=1207.939,-65.789,-39.589,179.652,5.480,149.065
C06053=1207.944,-66.039,-39.578,179.650,5.480,149.065
C06054=1207.949,-66.289,-39.566,179.647,5.480,149.066
C06055=1207.954,-66.538,-39.555,179.644,5.479,149.067
C06056=1207.959,-66.788,-39.543,179.642,5.479,149.067
C06057=1207.965,-67.037,-39.532,179.640,5.479,149.068
C06058=1207.969,-67.287,-39.521,179.638,5.479,149.069
C06059=1207.975,-67.537,-39.509,179.635,5.479,149.069
C06060=1207.980,-67.787,-39.498,179.633,5.478,149.070
C06061=1207.985,-68.037,-39.486,179.631,5.478,149.071
C06062=1207.990,-68.286,-39.475,179.628,5.478,149.071
C06063=1207.996,-68.536,-39.463,179.626,5.478,149.072
C06064=1208.001,-68.785,-39.452,179.623,5.478,149.073
C06065=1208.005,-69.035,-39.441,179.620,5.478,149.074
C06066=1208.011,-69.284,-39.429,179.619,5.477,149.074
C06067=1208.016,-69.535,-39.419,179.616,5.477,149.075
C06068=1208.022,-69.785,-39.407,179.614,5.477,149.075
C06069=1208.026,-70.034,-39.396,179.611,5.477,149.076
C06070=1208.032,-70.283,-39.385,179.609,5.477,149.077
C06071=1208.037,-70.533,-39.373,179.607,5.477,149.078
C06072=1208.042,-70.783,-39.362,179.605,5.476,149.078
C06073=1208.048,-71.032,-39.351,179.602,5.476,149.079
C06074=1208.053,-71.282,-39.339,179.600,5.476,149.079
C06075=1208.058,-71.532,-39.328,179.598,5.476,149.080
C06076=1208.063,-71.782,-39.317,179.595,5.476,149.081
C06077=1208.069,-72.031,-39.306,179.592,5.475,149.082
C06078=1208.073,-72.281,-39.295,179.590,5.476,149.082
C06079=1208.079,-72.531,-39.283,179.588,5.475,149.083
C06080=1208.084,-72.780,-39.273,179.586,5.475,149.084
C06081=1208.089,-73.030,-39.261,179.583,5.475,149.084
C06082=1208.094,-73.280,-39.249,179.581,5.474,149.085
C06083=1208.099,-73.530,-39.238,179.579,5.475,149.086
C06084=1208.105,-73.779,-39.228,179.576,5.474,149.086
C06085=1208.110,-74.029,-39.216,179.574,5.475,149.087
C06086=1208.115,-74.279,-39.205,179.572,5.474,149.088
C06087=1208.120,-74.528,-39.195,179.570,5.474,149.088
C06088=1208.126,-74.799,-39.182,179.567,5.474,149.089
C06089=1208.132,-75.070,-39.170,179.564,5.473,149.090
C06090=1208.138,-75.340,-39.158,179.562,5.473,149.090
C06091=1208.143,-75.611,-39.145,179.559,5.474,149.091
C06092=1208.148,-75.861,-39.135,179.557,5.473,149.092
C06093=1208.153,-76.110,-39.124,179.555,5.473,149.092
C06094=1208.158,-76.360,-39.113,179.552,5.473,149.093
C06095=1208.165,-76.609,-39.102,179.549,5.472,149.094
C06096=1208.169,-76.859,-39.090,179.547,5.473,149.095
C06097=1208.174,-77.109,-39.080,179.545,5.472,149.095
C06098=1208.179,-77.358,-39.069,179.543,5.472,149.096
C06099=1208.185,-77.609,-39.058,179.540,5.472,149.097
C06100=1208.190,-77.858,-39.046,179.538,5.472,149.097
C06101=1208.195,-78.107,-39.035,179.536,5.472,149.098
C06102=1208.200,-78.358,-39.025,179.533,5.472,149.099
C06103=1208.206,-78.607,-39.013,179.531,5.472,149.099
C06104=1208.211,-78.857,-39.003,179.529,5.471,149.100
C06105=1208.216,-79.107,-38.992,179.527,5.471,149.101
C06106=1208.222,-79.356,-38.981,179.524,5.471,149.101
C06107=1208.226,-79.606,-38.970,179.522,5.471,149.102
C06108=1208.232,-79.856,-38.959,179.519,5.471,149.103
C06109=1208.237,-80.105,-38.948,179.517,5.471,149.103
C06110=1208.242,-80.356,-38.937,179.515,5.470,149.104
C06111=1208.248,-80.604,-38.926,179.512,5.470,149.105
C06112=1208.252,-80.854,-38.915,179.510,5.470,149.105
C06113=1208.258,-81.105,-38.904,179.507,5.470,149.106
C06114=1208.264,-81.354,-38.894,179.505,5.470,149.107
C06115=1208.268,-81.604,-38.882,179.503,5.470,149.107
C06116=1208.274,-81.853,-38.872,179.501,5.470,149.108
C06117=1208.279,-82.103,-38.861,179.498,5.469,149.109
C06118=1208.284,-82.353,-38.850,179.496,5.470,149.109
C06119=1208.290,-82.602,-38.839,179.494,5.469,149.110
C06120=1208.295,-82.853,-38.828,179.491,5.469,149.111
C06121=1208.300,-83.102,-38.817,179.489,5.469,149.111
C06122=1208.305,-83.352,-38.807,179.487,5.468,149.112
C06123=1208.310,-83.601,-38.796,179.485,5.469,149.113
C06124=1208.315,-83.851,-38.785,179.482,5.468,149.113
C06125=1208.320,-84.101,-38.775,179.480,5.469,149.114
C06126=1208.325,-84.350,-38.764,179.477,5.468,149.115
C06127=1208.330,-84.600,-38.753,179.476,5.468,149.115
C06128=1208.336,-84.850,-38.742,179.473,5.468,149.116
C06129=1208.341,-85.100,-38.731,179.471,5.468,149.117
C06130=1208.347,-85.349,-38.721,179.468,5.468,149.117
C06131=1208.352,-85.599,-38.710,179.465,5.467,149.118
C06132=1208.357,-85.849,-38.699,179.464,5.467,149.119
C06133=1208.362,-86.098,-38.688,179.461,5.467,149.119
C06134=1208.367,-86.349,-38.678,179.459,5.467,149.120
C06135=1208.373,-86.598,-38.667,179.456,5.467,149.121
C06136=1208.377,-86.848,-38.656,179.454,5.467,149.121
C06137=1208.383,-87.097,-38.646,179.452,5.467,149.122
C06138=1208.388,-87.347,-38.635,179.450,5.467,149.123
C06139=1208.393,-87.596,-38.624,179.447,5.466,149.123
C06140=1208.398,-87.847,-38.614,179.445,5.467,149.124
C06141=1208.404,-88.096,-38.604,179.443,5.466,149.125
C06142=1208.409,-88.346,-38.593,179.440,5.466,149.125
C06143=1208.414,-88.595,-38.582,179.438,5.466,149.126
C06144=1208.419,-88.846,-38.571,179.436,5.465,149.127
C06145=1208.425,-89.095,-38.561,179.434,5.466,149.127
C06146=1208.429,-89.345,-38.550,179.431,5.465,149.128
C06147=1208.435,-89.594,-38.540,179.429,5.466,149.129
C06148=1208.440,-89.845,-38.529,179.427,5.465,149.129
C06149=1208.446,-90.094,-38.519,179.425,5.465,149.130
C06150=1208.450,-90.344,-38.508,179.422,5.465,149.131
C06151=1208.456,-90.593,-38.498,179.420,5.465,149.131
C06152=1208.461,-90.843,-38.487,179.417,5.465,149.132
C06153=1208.466,-91.093,-38.477,179.416,5.465,149.133
C06154=1208.472,-91.343,-38.467,179.413,5.464,149.133
C06155=1208.477,-91.592,-38.455,179.411,5.465,149.134
C06156=1208.482,-91.842,-38.445,179.408,5.464,149.135
C06157=1208.487,-92.092,-38.434,179.405,5.464,149.135
C06158=1208.493,-92.342,-38.424,179.404,5.464,149.136
C06159=1208.498,-92.592,-38.414,179.401,5.463,149.137
C06160=1208.503,-92.841,-38.403,179.399,5.464,149.137
C06161=1208.509,-93.090,-38.393,179.396,5.463,149.138
C06162=1208.514,-93.341,-38.382,179.394,5.464,149.139
C06163=1208.519,-93.590,-38.372,179.392,5.463,149.139
C06164=1208.524,-93.840,-38.361,179.390,5.463,149.140
C06165=1208.530,-94.090,-38.351,179.387,5.463,149.141
C06166=1208.535,-94.340,-38.340,179.385,5.463,149.141
C06167=1208.540,-94.589,-38.330,179.383,5.463,149.142
C06168=1208.545,-94.838,-38.320,179.381,5.463,149.143
C06169=1208.550,-95.088,-38.309,179.378,5.462,149.143
C06170=1208.556,-95.338,-38.299,179.376,5.463,149.144
C06171=1208.561,-95.588,-38.288,179.374,5.462,149.145
C06172=1208.566,-95.838,-38.278,179.371,5.463,149.145
C06173=1208.572,-96.087,-38.268,179.369,5.462,149.146
C06174=1208.577,-96.338,-38.257,179.367,5.462,149.147
C06175=1208.583,-96.587,-38.247,179.365,5.462,149.147
C06176=1208.587,-96.837,-38.237,179.362,5.462,149.148
C06177=1208.592,-97.087,-38.227,179.360,5.462,149.149
C06178=1208.598,-97.336,-38.216,179.358,5.462,149.149
C06179=1208.603,-97.586,-38.206,179.355,5.461,149.150
C06180=1208.608,-97.835,-38.195,179.353,5.461,149.151
C06181=1208.614,-98.085,-38.185,179.351,5.461,149.151
C06182=1208.619,-98.335,-38.175,179.349,5.461,149.152
C06183=1208.624,-98.584,-38.165,179.346,5.461,149.153
C06184=1208.629,-98.835,-38.154,179.344,5.461,149.153
C06185=1208.634,-99.084,-38.144,179.342,5.461,149.154
C06186=1208.640,-99.334,-38.134,179.339,5.461,149.155
C06187=1208.645,-99.584,-38.123,179.337,5.461,149.155
C06188=1208.650,-99.833,-38.114,179.335,5.460,149.156
C06189=1208.655,-100.083,-38.104,179.333,5.460,149.157
C06190=1208.660,-100.333,-38.093,179.330,5.460,149.157
C06191=1208.666,-100.583,-38.083,179.328,5.460,149.158
C06192=1208.672,-100.854,-38.073,179.326,5.460,149.159
C06193=1208.678,-101.125,-38.061,179.324,5.460,149.159
C06194=1208.683,-101.397,-38.050,179.321,5.460,149.160
C06195=1208.688,-101.668,-38.040,179.318,5.459,149.161
C06196=1208.694,-101.917,-38.029,179.316,5.460,149.161
C06197=1208.699,-102.168,-38.019,179.313,5.459,149.162
C06198=1208.705,-102.417,-38.009,179.311,5.460,149.163
C06199=1208.709,-102.666,-37.999,179.309,5.459,149.164
C06200=1208.715,-102.916,-37.989,179.307,5.459,149.164
C06201=1208.720,-103.166,-37.978,179.304,5.459,149.165
C06202=1208.726,-103.416,-37.968,179.302,5.459,149.165
C06203=1208.731,-103.666,-37.959,179.300,5.459,149.166
C06204=1208.736,-103.916,-37.948,179.298,5.459,149.167
C06205=1208.741,-104.165,-37.938,179.295,5.458,149.167
C06206=1208.746,-104.415,-37.929,179.293,5.459,149.168
C06207=1208.751,-104.665,-37.918,179.291,5.458,149.169
C06208=1208.757,-104.914,-37.908,179.289,5.458,149.169
C06209=1208.762,-105.164,-37.898,179.286,5.458,149.170
C06210=1208.768,-105.414,-37.889,179.284,5.458,149.171
C06211=1208.773,-105.664,-37.878,179.282,5.458,149.171
C06212=1208.778,-105.914,-37.868,179.280,5.458,149.172
C06213=1208.783,-106.163,-37.858,179.277,5.457,149.173
C06214=1208.789,-106.412,-37.848,179.275,5.458,149.173
C06215=1208.794,-106.663,-37.838,179.273,5.457,149.174
C06216=1208.799,-106.913,-37.829,179.271,5.457,149.174
C06217=1208.804,-107.162,-37.818,179.268,5.457,149.175
C06218=1208.810,-107.412,-37.808,179.266,5.457,149.176
C06219=1208.814,-107.662,-37.798,179.263,5.457,149.177
C06220=1208.820,-107.912,-37.789,179.262,5.457,149.177
C06221=1208.826,-108.161,-37.779,179.259,5.456,149.178
C06222=1208.831,-108.410,-37.769,179.257,5.457,149.179
C06223=1208.836,-108.661,-37.758,179.254,5.456,149.179
C06224=1208.841,-108.911,-37.750,179.253,5.456,149.180
C06225=1208.846,-109.160,-37.739,179.250,5.456,149.180
C06226=1208.852,-109.410,-37.729,179.248,5.456,149.181
C06227=1208.856,-109.660,-37.719,179.245,5.456,149.182
C06228=1208.862,-109.910,-37.710,179.244,5.456,149.182
C06229=1208.868,-110.159,-37.699,179.241,5.456,149.183
C06230=1208.873,-110.409,-37.690,179.239,5.456,149.184
C06231=1208.879,-110.659,-37.680,179.236,5.456,149.185
C06232=1208.883,-110.909,-37.670,179.235,5.456,149.185
C06233=1208.888,-111.158,-37.660,179.233,5.456,149.186
C06234=1208.894,-111.408,-37.651,179.230,5.456,149.186
C06235=1208.899,-111.658,-37.641,179.228,5.456,149.187
C06236=1208.905,-111.907,-37.631,179.226,5.455,149.188
C06237=1208.909,-112.158,-37.622,179.224,5.456,149.188
C06238=1208.915,-112.407,-37.611,179.221,5.455,149.189
C06239=1208.920,-112.656,-37.602,179.219,5.455,149.190
C06240=1208.926,-112.907,-37.592,179.217,5.455,149.190
C06241=1208.931,-113.156,-37.583,179.215,5.455,149.191
C06242=1208.936,-113.405,-37.572,179.212,5.455,149.192
C06243=1208.941,-113.656,-37.563,179.210,5.455,149.192
C06244=1208.946,-113.905,-37.553,179.208,5.454,149.193
C06245=1208.952,-114.156,-37.543,179.206,5.455,149.194
C06246=1208.957,-114.405,-37.534,179.203,5.454,149.194
C06247=1208.963,-114.654,-37.524,179.201,5.454,149.195
C06248=1208.968,-114.904,-37.515,179.199,5.454,149.196
C06249=1208.973,-115.154,-37.505,179.196,5.454,149.196
C06250=1208.978,-115.404,-37.495,179.194,5.453,149.197
C06251=1208.984,-115.654,-37.485,179.192,5.454,149.197
C06252=1208.989,-115.904,-37.476,179.190,5.453,149.198
C06253=1208.994,-116.153,-37.466,179.187,5.454,149.199
C06254=1209.000,-116.403,-37.457,179.185,5.453,149.199
C06255=1209.005,-116.653,-37.447,179.183,5.453,149.200
C06256=1209.010,-116.902,-37.437,179.180,5.453,149.201
C06257=1209.015,-117.153,-37.427,179.179,5.453,149.201
C06258=1209.020,-117.402,-37.418,179.177,5.453,149.202
C06259=1209.025,-117.652,-37.409,179.174,5.453,149.203
C06260=1209.031,-117.901,-37.399,179.172,5.453,149.203
C06261=1209.036,-118.151,-37.390,179.170,5.453,149.204
C06262=1209.042,-118.401,-37.380,179.168,5.453,149.205
C06263=1209.047,-118.651,-37.371,179.165,5.453,149.205
C06264=1209.052,-118.900,-37.360,179.163,5.453,149.206
C06265=1209.058,-119.150,-37.352,179.161,5.452,149.207
C06266=1209.063,-119.401,-37.342,179.159,5.453,149.207
C06267=1209.068,-119.650,-37.332,179.156,5.452,149.208
C06268=1209.073,-119.900,-37.323,179.154,5.452,149.208
C06269=1209.079,-120.150,-37.313,179.152,5.452,149.209
C06270=1209.084,-120.399,-37.304,179.150,5.452,149.210
C06271=1209.089,-120.649,-37.294,179.147,5.451,149.210
C06272=1209.095,-120.899,-37.285,179.145,5.452,149.211
C06273=1209.099,-121.148,-37.275,179.143,5.451,149.212
C06274=1209.105,-121.398,-37.266,179.141,5.451,149.212
C06275=1209.110,-121.648,-37.257,179.139,5.452,149.213
C06276=1209.116,-121.898,-37.247,179.136,5.451,149.214
C06277=1209.121,-122.147,-37.238,179.135,5.451,149.214
C06278=1209.126,-122.397,-37.228,179.132,5.451,149.215
C06279=1209.132,-122.647,-37.219,179.130,5.451,149.216
C06280=1209.137,-122.897,-37.210,179.127,5.451,149.216
C06281=1209.141,-123.147,-37.200,179.126,5.451,149.217
C06282=1209.147,-123.397,-37.190,179.123,5.451,149.218
C06283=1209.152,-123.647,-37.181,179.121,5.451,149.218
C06284=1209.157,-123.896,-37.172,179.119,5.450,149.219
C06285=1209.163,-124.146,-37.162,179.117,5.451,149.219
C06286=1209.168,-124.396,-37.153,179.114,5.450,149.220
C06287=1209.173,-124.645,-37.144,179.112,5.450,149.221
C06288=1209.179,-124.895,-37.134,179.110,5.451,149.221
C06289=1209.184,-125.145,-37.125,179.108,5.450,149.222
C06290=1209.189,-125.394,-37.116,179.106,5.450,149.223
C06291=1209.195,-125.645,-37.106,179.103,5.450,149.223
C06292=1209.200,-125.894,-37.097,179.101,5.450,149.224
C06293=1209.205,-126.144,-37.088,179.099,5.449,149.225
C06294=1209.211,-126.394,-37.078,179.097,5.450,149.225
C06295=1209.216,-126.644,-37.069,179.094,5.449,149.226
C06296=1208.795,-126.654,-37.107,179.090,5.453,149.228
C06297=1208.789,-126.404,-37.116,179.093,5.453,149.227
C06298=1208.784,-126.154,-37.125,179.095,5.453,149.227
C06299=1208.779,-125.905,-37.135,179.097,5.453,149.226
C06300=1208.774,-125.655,-37.144,179.099,5.453,149.225
C06301=1208.768,-125.405,-37.153,179.102,5.454,149.225
C06302=1208.763,-125.156,-37.163,179.104,5.453,149.224
C06303=1208.758,-124.906,-37.172,179.106,5.454,149.223
C06304=1208.752,-124.656,-37.181,179.108,5.454,149.223
C06305=1208.748,-124.407,-37.191,179.110,5.453,149.222
C06306=1208.742,-124.156,-37.200,179.113,5.454,149.221
C06307=1208.736,-123.907,-37.209,179.114,5.454,149.221
C06308=1208.732,-123.657,-37.219,179.117,5.454,149.220
C06309=1208.726,-123.407,-37.228,179.119,5.454,149.219
C06310=1208.721,-123.157,-37.237,179.121,5.455,149.219
C06311=1208.716,-122.908,-37.247,179.123,5.454,149.218
C06312=1208.710,-122.658,-37.256,179.126,5.455,149.218
C06313=1208.705,-122.408,-37.265,179.128,5.455,149.217
C06314=1208.699,-122.158,-37.275,179.130,5.455,149.216
C06315=1208.694,-121.909,-37.284,179.132,5.455,149.216
C06316=1208.689,-121.659,-37.294,179.135,5.455,149.215
C06317=1208.683,-121.409,-37.303,179.137,5.455,149.214
C06318=1208.678,-121.159,-37.312,179.139,5.455,149.214
C06319=1208.673,-120.910,-37.322,179.141,5.455,149.213
C06320=1208.668,-120.659,-37.332,179.143,5.455,149.212
C06321=1208.663,-120.410,-37.341,179.146,5.455,149.212
C06322=1208.657,-120.160,-37.351,179.148,5.455,149.211
C06323=1208.652,-119.910,-37.360,179.150,5.456,149.211
C06324=1208.647,-119.661,-37.369,179.152,5.455,149.210
C06325=1208.641,-119.411,-37.379,179.155,5.456,149.209
C06326=1208.636,-119.161,-37.389,179.156,5.456,149.209
C06327=1208.630,-118.911,-37.398,179.159,5.456,149.208
C06328=1208.625,-118.662,-37.408,179.161,5.456,149.207
C06329=1208.620,-118.412,-37.417,179.164,5.456,149.206
C06330=1208.615,-118.163,-37.427,179.165,5.456,149.206
C06331=1208.610,-117.912,-37.436,179.168,5.457,149.205
C06332=1208.605,-117.663,-37.446,179.170,5.456,149.205
C06333=1208.599,-117.413,-37.455,179.172,5.457,149.204
C06334=1208.594,-117.163,-37.465,179.174,5.457,149.203
C06335=1208.589,-116.913,-37.474,179.177,5.457,149.203
C06336=1208.583,-116.664,-37.484,179.179,5.457,149.202
C06337=1208.578,-116.414,-37.493,179.181,5.457,149.201
C06338=1208.572,-116.164,-37.504,179.183,5.457,149.201
C06339=1208.568,-115.914,-37.513,179.186,5.457,149.200
C06340=1208.562,-115.664,-37.523,179.188,5.457,149.200
C06341=1208.557,-115.414,-37.532,179.190,5.457,149.199
C06342=1208.551,-115.165,-37.542,179.193,5.457,149.198
C06343=1208.546,-114.916,-37.552,179.194,5.457,149.198
C06344=1208.541,-114.665,-37.561,179.197,5.458,149.197
C06345=1208.536,-114.416,-37.571,179.199,5.457,149.196
C06346=1208.530,-114.165,-37.581,179.202,5.458,149.195
C06347=1208.525,-113.916,-37.590,179.203,5.458,149.195
C06348=1208.520,-113.667,-37.601,179.206,5.458,149.194
C06349=1208.515,-113.417,-37.609,179.208,5.458,149.194
C06350=1208.509,-113.167,-37.620,179.211,5.458,149.193
C06351=1208.504,-112.917,-37.629,179.212,5.458,149.192
C06352=1208.498,-112.668,-37.639,179.215,5.459,149.192
C06353=1208.493,-112.418,-37.649,179.217,5.458,149.191
C06354=1208.488,-112.168,-37.658,179.219,5.459,149.190
C06355=1208.483,-111.918,-37.668,179.221,5.459,149.190
C06356=1208.478,-111.669,-37.678,179.224,5.459,149.189
C06357=1208.472,-111.419,-37.688,179.226,5.459,149.188
C06358=1208.468,-111.169,-37.698,179.228,5.459,149.188
C06359=1208.462,-110.919,-37.708,179.230,5.459,149.187
C06360=1208.456,-110.669,-37.717,179.233,5.460,149.186
C06361=1208.451,-110.420,-37.727,179.235,5.459,149.186
C06362=1208.446,-110.170,-37.737,179.237,5.459,149.185
C06363=1208.441,-109.920,-37.746,179.239,5.460,149.184
C06364=1208.435,-109.670,-37.757,179.241,5.459,149.184
C06365=1208.430,-109.421,-37.767,179.244,5.460,149.183
C06366=1208.425,-109.171,-37.776,179.246,5.460,149.183
C06367=1208.419,-108.921,-37.786,179.248,5.460,149.182
C06368=1208.415,-108.671,-37.796,179.250,5.460,149.181
C06369=1208.409,-108.422,-37.806,179.253,5.460,149.181
C06370=1208.403,-108.172,-37.816,179.255,5.460,149.180
C06371=1208.398,-107.922,-37.825,179.257,5.460,149.179
C06372=1208.393,-107.672,-37.836,179.260,5.460,149.178
C06373=1208.388,-107.423,-37.846,179.262,5.461,149.178
C06374=1208.383,-107.173,-37.855,179.264,5.460,149.177
C06375=1208.377,-106.923,-37.865,179.266,5.461,149.177
C06376=1208.372,-106.673,-37.876,179.269,5.460,149.176
C06377=1208.367,-106.424,-37.885,179.271,5.461,149.175
C06378=1208.362,-106.174,-37.895,179.273,5.461,149.175
C06379=1208.356,-105.924,-37.905,179.276,5.461,149.174
C06380=1208.351,-105.674,-37.915,179.278,5.461,149.173
C06381=1208.346,-105.425,-37.925,179.280,5.462,149.173
C06382=1208.340,-105.175,-37.935,179.282,5.461,149.172
C06383=1208.335,-104.926,-37.945,179.285,5.462,149.171
C06384=1208.330,-104.676,-37.956,179.287,5.461,149.171
C06385=1208.325,-104.425,-37.965,179.289,5.462,149.170
C06386=1208.320,-104.176,-37.975,179.291,5.462,149.169
C06387=1208.315,-103.926,-37.985,179.294,5.462,149.169
C06388=1208.309,-103.676,-37.995,179.296,5.462,149.168
C06389=1208.304,-103.427,-38.005,179.298,5.463,149.168
C06390=1208.299,-103.178,-38.015,179.300,5.462,149.167
C06391=1208.294,-102.927,-38.026,179.303,5.463,149.166
C06392=1208.288,-102.678,-38.036,179.305,5.462,149.165
C06393=1208.283,-102.428,-38.045,179.307,5.463,149.165
C06394=1208.278,-102.178,-38.055,179.309,5.463,149.164
C06395=1208.272,-101.928,-38.066,179.312,5.463,149.163
C06396=1208.267,-101.679,-38.076,179.314,5.463,149.163
C06397=1208.261,-101.407,-38.087,179.316,5.463,149.162
C06398=1208.256,-101.136,-38.098,179.319,5.464,149.161
C06399=1208.250,-100.864,-38.109,179.321,5.463,149.161
C06400=1208.245,-100.594,-38.120,179.324,5.464,149.160
C06401=1208.240,-100.344,-38.130,179.326,5.463,149.159
C06402=1208.234,-100.094,-38.141,179.328,5.464,149.159
C06403=1208.228,-99.845,-38.151,179.330,5.464,149.158
C06404=1208.224,-99.595,-38.161,179.333,5.464,149.157
C06405=1208.219,-99.345,-38.171,179.335,5.464,149.157
C06406=1208.213,-99.096,-38.181,179.337,5.464,149.156
C06407=1208.208,-98.845,-38.192,179.340,5.465,149.155
C06408=1208.202,-98.596,-38.202,179.342,5.465,149.155
C06409=1208.197,-98.346,-38.212,179.345,5.465,149.154
C06410=1208.192,-98.096,-38.222,179.347,5.465,149.153
C06411=1208.187,-97.847,-38.232,179.349,5.465,149.153
C06412=1208.181,-97.597,-38.243,179.351,5.465,149.152
C06413=1208.176,-97.347,-38.253,179.354,5.465,149.151
C06414=1208.171,-97.097,-38.263,179.356,5.465,149.151
C06415=1208.166,-96.847,-38.274,179.358,5.466,149.150
C06416=1208.161,-96.598,-38.284,179.360,5.465,149.149
C06417=1208.155,-96.348,-38.294,179.363,5.466,149.149
C06418=1208.150,-96.098,-38.304,179.365,5.466,149.148
C06419=1208.145,-95.849,-38.315,179.368,5.466,149.147
C06420=1208.140,-95.598,-38.325,179.369,5.466,149.147
C06421=1208.134,-95.349,-38.335,179.372,5.466,149.146
C06422=1208.128,-95.099,-38.346,179.374,5.466,149.145
C06423=1208.123,-94.849,-38.356,179.377,5.466,149.145
C06424=1208.118,-94.600,-38.367,179.379,5.466,149.144
C06425=1208.114,-94.350,-38.377,179.381,5.467,149.143
C06426=1208.108,-94.101,-38.387,179.383,5.466,149.143
C06427=1208.103,-93.851,-38.398,179.386,5.467,149.142
C06428=1208.098,-93.601,-38.408,179.388,5.467,149.141
C06429=1208.092,-93.351,-38.418,179.390,5.467,149.141
C06430=1208.087,-93.101,-38.429,179.392,5.467,149.140
C06431=1208.082,-92.852,-38.440,179.395,5.467,149.139
C06432=1208.077,-92.602,-38.450,179.397,5.468,149.139
C06433=1208.071,-92.352,-38.461,179.399,5.467,149.138
C06434=1208.066,-92.103,-38.471,179.402,5.468,149.138
C06435=1208.061,-91.853,-38.481,179.404,5.468,149.137
C06436=1208.055,-91.603,-38.492,179.406,5.468,149.136
C06437=1208.050,-91.353,-38.503,179.408,5.468,149.135
C06438=1208.045,-91.104,-38.513,179.411,5.468,149.135
C06439=1208.040,-90.854,-38.524,179.413,5.468,149.134
C06440=1208.034,-90.604,-38.534,179.415,5.469,149.133
C06441=1208.029,-90.354,-38.545,179.417,5.468,149.133
C06442=1208.024,-90.105,-38.555,179.420,5.469,149.132
C06443=1208.019,-89.855,-38.566,179.422,5.468,149.131
C06444=1208.013,-89.605,-38.576,179.424,5.469,149.131
C06445=1208.009,-89.355,-38.587,179.426,5.469,149.130
C06446=1208.003,-89.106,-38.598,179.429,5.469,149.129
C06447=1207.997,-88.856,-38.608,179.432,5.470,149.129
C06448=1207.992,-88.606,-38.618,179.434,5.469,149.128
C06449=1207.987,-88.357,-38.629,179.436,5.470,149.128
C06450=1207.982,-88.107,-38.640,179.438,5.470,149.127
C06451=1207.976,-87.857,-38.650,179.441,5.470,149.126
C06452=1207.971,-87.607,-38.661,179.443,5.470,149.125
C06453=1207.966,-87.358,-38.672,179.446,5.470,149.125
C06454=1207.961,-87.108,-38.682,179.448,5.470,149.124
C06455=1207.956,-86.858,-38.693,179.450,5.471,149.123
C06456=1207.951,-86.609,-38.704,179.452,5.470,149.123
C06457=1207.946,-86.359,-38.714,179.455,5.471,149.122
C06458=1207.940,-86.109,-38.724,179.457,5.470,149.121
C06459=1207.936,-85.859,-38.736,179.459,5.471,149.121
C06460=1207.930,-85.610,-38.746,179.462,5.472,149.120
C06461=1207.925,-85.360,-38.757,179.464,5.471,149.119
C06462=1207.920,-85.111,-38.767,179.466,5.472,149.119
C06463=1207.915,-84.860,-38.778,179.468,5.471,149.118
C06464=1207.909,-84.612,-38.789,179.471,5.472,149.117
C06465=1207.904,-84.361,-38.800,179.473,5.472,149.117
C06466=1207.898,-84.111,-38.810,179.475,5.472,149.116
C06467=1207.893,-83.862,-38.822,179.477,5.472,149.115
C06468=1207.888,-83.612,-38.832,179.480,5.472,149.115
C06469=1207.883,-83.363,-38.843,179.482,5.472,149.114
C06470=1207.878,-83.112,-38.854,179.485,5.472,149.113
C06471=1207.873,-82.863,-38.865,179.487,5.473,149.113
C06472=1207.868,-82.613,-38.875,179.489,5.473,149.112
C06473=1207.862,-82.364,-38.885,179.492,5.473,149.111
C06474=1207.857,-82.114,-38.897,179.494,5.473,149.111
C06475=1207.852,-81.863,-38.908,179.497,5.473,149.110
C06476=1207.846,-81.615,-38.919,179.498,5.473,149.110
C06477=1207.841,-81.364,-38.929,179.501,5.474,149.109
C06478=1207.836,-81.115,-38.940,179.503,5.473,149.108
C06479=1207.831,-80.865,-38.951,179.506,5.474,149.107
C06480=1207.826,-80.616,-38.962,179.508,5.474,149.107
C06481=1207.820,-80.366,-38.973,179.510,5.474,149.106
C06482=1207.815,-80.116,-38.984,179.513,5.475,149.105
C06483=1207.810,-79.867,-38.994,179.515,5.474,149.105
C06484=1207.805,-79.617,-39.006,179.517,5.475,149.104
C06485=1207.800,-79.367,-39.016,179.519,5.474,149.103
C06486=1207.794,-79.117,-39.028,179.522,5.475,149.103
C06487=1207.789,-78.867,-39.038,179.525,5.475,149.102
C06488=1207.784,-78.618,-39.049,179.526,5.475,149.101
C06489=1207.779,-78.369,-39.061,179.529,5.476,149.101
C06490=1207.774,-78.118,-39.071,179.531,5.475,149.100
C06491=1207.768,-77.869,-39.083,179.534,5.476,149.099
C06492=1207.763,-77.619,-39.093,179.536,5.475,149.099
C06493=1207.758,-77.369,-39.105,179.539,5.476,149.098
C06494=1207.753,-77.120,-39.115,179.540,5.476,149.097
C06495=1207.747,-76.870,-39.127,179.543,5.476,149.097
C06496=1207.742,-76.621,-39.138,179.545,5.477,149.096
C06497=1207.737,-76.371,-39.148,179.548,5.476,149.095
C06498=1207.732,-76.121,-39.160,179.550,5.477,149.095
C06499=1207.726,-75.872,-39.171,179.552,5.476,149.094
C06500=1207.721,-75.621,-39.182,179.555,5.477,149.093
C06501=1207.716,-75.351,-39.194,179.557,5.478,149.093
C06502=1207.710,-75.080,-39.206,179.560,5.477,149.092
C06503=1207.705,-74.810,-39.217,179.562,5.477,149.091
C06504=1207.699,-74.539,-39.230,179.565,5.478,149.090
C06505=1207.693,-74.289,-39.241,179.567,5.477,149.090
C06506=1207.688,-74.040,-39.252,179.569,5.478,149.089
C06507=1207.683,-73.789,-39.263,179.571,5.478,149.088
C06508=1207.678,-73.541,-39.274,179.574,5.478,149.088
C06509=1207.673,-73.291,-39.286,179.577,5.479,149.087
C06510=1207.668,-73.041,-39.297,179.579,5.478,149.086
C06511=1207.662,-72.791,-39.307,179.582,5.479,149.086
C06512=1207.657,-72.542,-39.319,179.583,5.479,149.085
C06513=1207.652,-72.292,-39.331,179.586,5.479,149.084
C06514=1207.647,-72.041,-39.342,179.588,5.480,149.084
C06515=1207.641,-71.792,-39.353,179.591,5.479,149.083
C06516=1207.637,-71.543,-39.364,179.593,5.480,149.082
C06517=1207.631,-71.293,-39.376,179.595,5.479,149.082
C06518=1207.626,-71.043,-39.386,179.598,5.480,149.081
C06519=1207.621,-70.794,-39.397,179.600,5.480,149.080
C06520=1207.615,-70.544,-39.409,179.602,5.480,149.080
C06521=1207.611,-70.294,-39.420,179.605,5.481,149.079
C06522=1207.605,-70.045,-39.432,179.607,5.480,149.078
C06523=1207.600,-69.795,-39.443,179.610,5.481,149.078
C06524=1207.595,-69.545,-39.454,179.612,5.481,149.077
C06525=1207.590,-69.295,-39.466,179.614,5.481,149.076
C06526=1207.584,-69.046,-39.477,179.617,5.482,149.076
C06527=1207.579,-68.796,-39.489,179.619,5.481,149.075
C06528=1207.574,-68.546,-39.499,179.621,5.482,149.074
C06529=1207.569,-68.296,-39.510,179.623,5.482,149.074
C06530=1207.563,-68.047,-39.522,179.626,5.482,149.073
C06531=1207.558,-67.797,-39.533,179.629,5.482,149.072
C06532=1207.553,-67.548,-39.545,179.630,5.482,149.072
C06533=1207.548,-67.298,-39.556,179.633,5.483,149.071
C06534=1207.542,-67.049,-39.568,179.635,5.483,149.070
C06535=1207.537,-66.798,-39.578,179.638,5.483,149.070
C06536=1207.532,-66.549,-39.590,179.641,5.483,149.069
C06537=1207.527,-66.299,-39.602,179.643,5.483,149.068
C06538=1207.522,-66.049,-39.613,179.645,5.483,149.067
C06539=1207.516,-65.800,-39.624,179.647,5.484,149.067
C06540=1207.512,-65.550,-39.636,179.650,5.484,149.066
C06541=1207.506,-65.300,-39.648,179.652,5.484,149.066
C06542=1207.502,-65.051,-39.659,179.654,5.484,149.065
C06543=1207.496,-64.801,-39.671,179.657,5.484,149.064
C06544=1207.491,-64.552,-39.682,179.659,5.484,149.063
C06545=1207.485,-64.302,-39.694,179.662,5.485,149.063
C06546=1207.481,-64.052,-39.705,179.664,5.485,149.062
C06547=1207.475,-63.802,-39.717,179.666,5.485,149.062
C06548=1207.471,-63.553,-39.728,179.669,5.486,149.061
C06549=1207.465,-63.303,-39.740,179.671,5.485,149.060
C06550=1207.460,-63.054,-39.751,179.673,5.486,149.059
C06551=1207.454,-62.804,-39.763,179.676,5.486,149.059
C06552=1207.449,-62.554,-39.775,179.678,5.486,149.058
C06553=1207.444,-62.304,-39.786,179.680,5.487,149.058
C06554=1207.439,-62.055,-39.798,179.682,5.486,149.057
C06555=1207.434,-61.805,-39.809,179.685,5.487,149.056
C06556=1207.428,-61.556,-39.821,179.688,5.487,149.055
C06557=1207.424,-61.306,-39.832,179.690,5.487,149.055
C06558=1207.418,-61.056,-39.844,179.692,5.487,149.054
C06559=1207.413,-60.807,-39.855,179.695,5.488,149.053
C06560=1207.408,-60.557,-39.867,179.697,5.488,149.053
C06561=1207.403,-60.307,-39.879,179.699,5.488,149.052
C06562=1207.398,-60.057,-39.890,179.701,5.488,149.051
C06563=1207.392,-59.807,-39.902,179.704,5.488,149.051
C06564=1207.387,-59.558,-39.913,179.707,5.489,149.050
C06565=1207.382,-59.308,-39.925,179.709,5.488,149.049
C06566=1207.377,-59.059,-39.937,179.712,5.489,149.049
C06567=1207.372,-58.809,-39.949,179.714,5.488,149.048
C06568=1207.366,-58.559,-39.961,179.716,5.489,149.047
C06569=1207.362,-58.310,-39.972,179.719,5.490,149.047
C06570=1207.356,-58.060,-39.984,179.721,5.489,149.046
C06571=1207.351,-57.810,-39.996,179.723,5.490,149.045
C06572=1207.346,-57.560,-40.007,179.726,5.490,149.045
C06573=1207.341,-57.310,-40.019,179.728,5.490,149.044
C06574=1207.336,-57.061,-40.031,179.731,5.490,149.043
C06575=1207.330,-56.812,-40.042,179.732,5.490,149.043
C06576=1207.325,-56.562,-40.054,179.735,5.491,149.042
C06577=1207.320,-56.312,-40.066,179.738,5.491,149.041
C06578=1207.315,-56.063,-40.077,179.740,5.491,149.041
C06579=1207.310,-55.813,-40.090,179.742,5.491,149.040
C06580=1207.304,-55.563,-40.102,179.745,5.492,149.039
C06581=1207.300,-55.314,-40.113,179.747,5.491,149.038
C06582=1207.294,-55.064,-40.125,179.750,5.492,149.038
C06583=1207.289,-54.814,-40.137,179.752,5.493,149.037
C06584=1207.284,-54.565,-40.149,179.754,5.492,149.037
C06585=1207.279,-54.315,-40.161,179.757,5.493,149.036
C06586=1207.273,-54.065,-40.173,179.759,5.492,149.035
C06587=1207.269,-53.815,-40.184,179.761,5.493,149.034
C06588=1207.264,-53.566,-40.197,179.764,5.493,149.034
C06589=1207.258,-53.316,-40.209,179.766,5.493,149.033
C06590=1207.253,-53.066,-40.220,179.769,5.493,149.032
C06591=1207.248,-52.817,-40.232,179.771,5.494,149.032
C06592=1207.243,-52.567,-40.244,179.773,5.494,149.031
C06593=1207.238,-52.317,-40.256,179.776,5.494,149.030
C06594=1207.232,-52.067,-40.268,179.778,5.495,149.030
C06595=1207.228,-51.818,-40.280,179.781,5.495,149.029
C06596=1207.222,-51.568,-40.292,179.783,5.495,149.028
C06597=1207.217,-51.318,-40.304,179.786,5.495,149.028
C06598=1207.212,-51.069,-40.316,179.788,5.495,149.027
C06599=1207.207,-50.819,-40.328,179.790,5.496,149.027
C06600=1207.202,-50.570,-40.340,179.792,5.496,149.026
C06601=1207.197,-50.320,-40.352,179.795,5.496,149.025
C06602=1207.191,-50.070,-40.364,179.798,5.497,149.024
C06603=1207.186,-49.821,-40.377,179.800,5.496,149.024
C06604=1207.181,-49.571,-40.388,179.802,5.497,149.023
C06605=1207.175,-49.301,-40.401,179.805,5.497,149.022
C06606=1207.169,-49.031,-40.414,179.808,5.498,149.022
C06607=1207.164,-48.761,-40.428,179.810,5.497,149.021
C06608=1207.158,-48.492,-40.440,179.812,5.498,149.020
C06609=1207.153,-48.242,-40.452,179.815,5.498,149.019
C06610=1207.148,-47.992,-40.465,179.818,5.499,149.019
C06611=1207.142,-47.742,-40.477,179.820,5.498,149.018
C06612=1207.139,-47.493,-40.489,179.822,5.499,149.017
C06613=1207.133,-47.243,-40.501,179.825,5.499,149.017
C06614=1207.128,-46.993,-40.513,179.827,5.499,149.016
C06615=1207.123,-46.744,-40.526,179.829,5.500,149.015
C06616=1207.117,-46.494,-40.537,179.832,5.500,149.015
C06617=1207.112,-46.244,-40.550,179.834,5.500,149.014
C06618=1207.107,-45.994,-40.562,179.837,5.500,149.013
C06619=1207.102,-45.745,-40.575,179.839,5.501,149.013
C06620=1207.097,-45.495,-40.586,179.842,5.500,149.012
C06621=1207.092,-45.246,-40.598,179.844,5.501,149.011
C06622=1207.086,-44.996,-40.610,179.847,5.501,149.011
C06623=1207.081,-44.747,-40.623,179.848,5.501,149.010
C06624=1207.076,-44.497,-40.635,179.851,5.502,149.009
C06625=1207.071,-44.248,-40.647,179.854,5.502,149.009
C06626=1207.066,-43.997,-40.660,179.856,5.502,149.008
C06627=1207.061,-43.748,-40.672,179.859,5.502,149.007
C06628=1207.056,-43.498,-40.685,179.861,5.503,149.007
C06629=1207.050,-43.248,-40.697,179.863,5.502,149.006
C06630=1207.045,-42.999,-40.709,179.866,5.503,149.005
C06631=1207.040,-42.749,-40.721,179.868,5.504,149.005
C06632=1207.034,-42.500,-40.734,179.870,5.503,149.004
C06633=1207.029,-42.250,-40.746,179.873,5.504,149.003
C06634=1207.024,-42.001,-40.758,179.876,5.504,149.003
C06635=1207.019,-41.750,-40.771,179.878,5.504,149.002
C06636=1207.015,-41.501,-40.783,179.880,5.504,149.001
C06637=1207.010,-41.252,-40.795,179.883,5.505,149.001
C06638=1207.004,-41.002,-40.808,179.885,5.505,149.000
C06639=1206.999,-40.752,-40.820,179.887,5.505,148.999
C06640=1206.994,-40.503,-40.832,179.890,5.506,148.999
C06641=1206.989,-40.254,-40.845,179.892,5.506,148.998
C06642=1206.984,-40.003,-40.857,179.895,5.506,148.997
C06643=1206.979,-39.754,-40.870,179.897,5.507,148.997
C06644=1206.974,-39.504,-40.882,179.899,5.506,148.996
C06645=1206.967,-39.254,-40.895,179.902,5.507,148.995
C06646=1206.962,-39.005,-40.907,179.905,5.507,148.994
C06647=1206.957,-38.756,-40.920,179.907,5.507,148.994
C06648=1206.952,-38.505,-40.932,179.909,5.508,148.993
C06649=1206.947,-38.256,-40.945,179.912,5.508,148.993
C06650=1206.942,-38.006,-40.957,179.914,5.509,148.992
C06651=1206.937,-37.757,-40.970,179.916,5.508,148.991
C06652=1206.932,-37.507,-40.982,179.919,5.509,148.990
C06653=1206.927,-37.257,-40.995,179.922,5.509,148.990
C06654=1206.922,-37.008,-41.008,179.924,5.509,148.989
C06655=1206.917,-36.758,-41.020,179.926,5.509,148.988
C06656=1206.911,-36.508,-41.032,179.929,5.510,148.988
C06657=1206.906,-36.259,-41.045,179.931,5.510,148.987
C06658=1206.902,-36.009,-41.058,179.933,5.510,148.987
C06659=1206.896,-35.759,-41.071,179.936,5.511,148.986
C06660=1206.890,-35.509,-41.083,179.939,5.511,148.985
C06661=1206.885,-35.260,-41.095,179.941,5.511,148.984
C06662=1206.880,-35.011,-41.108,179.943,5.511,148.984
C06663=1206.876,-34.761,-41.121,179.946,5.512,148.983
C06664=1206.871,-34.512,-41.133,179.948,5.511,148.982
C06665=1206.865,-34.262,-41.146,179.950,5.512,148.982
C06666=1206.860,-34.012,-41.158,179.953,5.513,148.981
C06667=1206.855,-33.762,-41.171,179.955,5.512,148.980
C06668=1206.850,-33.513,-41.184,179.958,5.513,148.980
C06669=1206.845,-33.263,-41.197,179.960,5.513,148.979
C06670=1206.839,-33.014,-41.209,179.963,5.514,148.978
C06671=1206.835,-32.764,-41.222,179.965,5.514,148.978
C06672=1206.830,-32.515,-41.235,179.968,5.514,148.977
C06673=1206.824,-32.265,-41.248,179.970,5.514,148.976
C06674=1206.818,-32.015,-41.260,179.972,5.514,148.976
C06675=1206.814,-31.765,-41.273,179.975,5.515,148.975
C06676=1206.809,-31.516,-41.285,179.977,5.515,148.974
C06677=1206.804,-31.266,-41.298,179.980,5.516,148.974
C06678=1206.798,-31.016,-41.312,179.982,5.516,148.973
C06679=1206.793,-30.767,-41.324,179.985,5.516,148.972
C06680=1206.788,-30.517,-41.337,179.987,5.517,148.972
C06681=1206.783,-30.268,-41.349,179.990,5.516,148.971
C06682=1206.779,-30.018,-41.362,179.992,5.517,148.970
C06683=1206.773,-29.769,-41.376,179.994,5.518,148.970
C06684=1206.768,-29.519,-41.388,179.997,5.518,148.969
C06685=1206.763,-29.269,-41.401,179.999,5.518,148.968
C06686=1206.758,-29.020,-41.414,-179.998,5.518,148.968
C06687=1206.752,-28.770,-41.427,-179.996,5.519,148.967
C06688=1206.748,-28.520,-41.440,-179.993,5.519,148.966
C06689=1206.742,-28.271,-41.453,-179.991,5.519,148.966
C06690=1206.737,-28.022,-41.465,-179.988,5.519,148.965
C06691=1206.732,-27.771,-41.479,-179.986,5.520,148.964
C06692=1206.727,-27.522,-41.491,-179.984,5.520,148.964
C06693=1206.722,-27.273,-41.504,-179.981,5.520,148.963
C06694=1206.717,-27.023,-41.517,-179.979,5.521,148.962
C06695=1206.711,-26.773,-41.530,-179.976,5.521,148.962
C06696=1206.706,-26.524,-41.543,-179.974,5.521,148.961
C06697=1206.702,-26.274,-41.556,-179.971,5.521,148.960
C06698=1206.696,-26.024,-41.569,-179.969,5.522,148.959
C06699=1206.691,-25.775,-41.581,-179.966,5.522,148.959
C06700=1206.687,-25.525,-41.595,-179.964,5.522,148.958
C06701=1206.681,-25.276,-41.608,-179.962,5.523,148.958
C06702=1206.676,-25.026,-41.621,-179.959,5.523,148.957
C06703=1206.671,-24.776,-41.634,-179.956,5.524,148.956
C06704=1206.665,-24.527,-41.647,-179.954,5.523,148.956
C06705=1206.661,-24.277,-41.660,-179.952,5.524,148.955
C06706=1206.656,-24.027,-41.673,-179.949,5.524,148.954
C06707=1206.650,-23.778,-41.687,-179.946,5.525,148.953
C06708=1206.645,-23.528,-41.700,-179.945,5.525,148.953
C06709=1206.639,-23.259,-41.713,-179.942,5.525,148.952
C06710=1206.634,-22.989,-41.727,-179.939,5.525,148.951
C06711=1206.629,-22.720,-41.742,-179.936,5.526,148.951
C06712=1206.624,-22.450,-41.756,-179.934,5.526,148.950
C06713=1206.618,-22.200,-41.769,-179.931,5.527,148.949
C06714=1206.613,-21.951,-41.782,-179.929,5.527,148.949
C06715=1206.608,-21.701,-41.796,-179.926,5.527,148.948
C06716=1206.603,-21.452,-41.808,-179.924,5.528,148.947
C06717=1206.598,-21.202,-41.821,-179.921,5.528,148.947
C06718=1206.592,-20.952,-41.835,-179.919,5.528,148.946
C06719=1206.587,-20.704,-41.848,-179.917,5.529,148.945
C06720=1206.582,-20.453,-41.862,-179.914,5.529,148.945
C06721=1206.577,-20.204,-41.874,-179.911,5.530,148.944
C06722=1206.572,-19.954,-41.888,-179.909,5.529,148.943
C06723=1206.567,-19.705,-41.901,-179.907,5.530,148.943
C06724=1206.562,-19.455,-41.915,-179.904,5.530,148.942
C06725=1206.557,-19.205,-41.927,-179.902,5.531,148.941
C06726=1206.552,-18.955,-41.940,-179.900,5.531,148.941
C06727=1206.546,-18.706,-41.954,-179.897,5.531,148.940
C06728=1206.542,-18.456,-41.967,-179.894,5.532,148.939
C06729=1206.536,-18.207,-41.980,-179.892,5.532,148.939
C06730=1206.531,-17.958,-41.993,-179.889,5.533,148.938
C06731=1206.526,-17.708,-42.007,-179.887,5.532,148.937
C06732=1206.521,-17.458,-42.020,-179.884,5.533,148.937
C06733=1206.516,-17.209,-42.034,-179.882,5.534,148.936
C06734=1206.511,-16.959,-42.047,-179.879,5.534,148.935
C06735=1206.506,-16.710,-42.061,-179.877,5.534,148.935
C06736=1206.501,-16.460,-42.073,-179.875,5.534,148.934
C06737=1206.495,-16.210,-42.087,-179.872,5.535,148.933
C06738=1206.491,-15.961,-42.100,-179.869,5.535,148.933
C06739=1206.485,-15.711,-42.114,-179.867,5.536,148.932
C06740=1206.480,-15.461,-42.127,-179.865,5.535,148.931
C06741=1206.475,-15.212,-42.141,-179.862,5.536,148.931
C06742=1206.469,-14.962,-42.154,-179.860,5.537,148.930
C06743=1206.465,-14.713,-42.168,-179.857,5.537,148.929
C06744=1206.459,-14.463,-42.181,-179.855,5.537,148.929
C06745=1206.455,-14.214,-42.194,-179.852,5.537,148.928
C06746=1206.449,-13.964,-42.208,-179.850,5.538,148.927
C06747=1206.444,-13.715,-42.222,-179.847,5.538,148.927
C06748=1206.440,-13.465,-42.235,-179.844,5.539,148.926
C06749=1206.434,-13.216,-42.249,-179.842,5.539,148.925
C06750=1206.430,-12.966,-42.262,-179.840,5.539,148.925
C06751=1206.424,-12.717,-42.276,-179.838,5.540,148.924
C06752=1206.420,-12.467,-42.289,-179.835,5.540,148.923
C06753=1206.414,-12.218,-42.303,-179.832,5.541,148.923
C06754=1206.409,-11.967,-42.316,-179.830,5.541,148.922
C06755=1206.404,-11.719,-42.329,-179.828,5.541,148.921
C06756=1206.399,-11.468,-42.343,-179.825,5.542,148.921
C06757=1206.394,-11.218,-42.357,-179.822,5.542,148.920
C06758=1206.389,-10.969,-42.370,-179.821,5.542,148.919
C06759=1206.384,-10.719,-42.384,-179.818,5.543,148.919
C06760=1206.378,-10.470,-42.397,-179.815,5.543,148.918
C06761=1206.374,-10.220,-42.411,-179.813,5.544,148.917
C06762=1206.368,-9.971,-42.424,-179.810,5.544,148.917
C06763=1206.363,-9.721,-42.439,-179.808,5.544,148.916
C06764=1206.359,-9.472,-42.452,-179.805,5.544,148.915
C06765=1206.353,-9.222,-42.465,-179.803,5.545,148.915
C06766=1206.348,-8.972,-42.480,-179.800,5.546,148.914
C06767=1206.343,-8.724,-42.493,-179.798,5.546,148.913
C06768=1206.338,-8.473,-42.507,-179.795,5.547,148.913
C06769=1206.333,-8.224,-42.521,-179.793,5.546,148.912
C06770=1206.328,-7.974,-42.533,-179.790,5.547,148.911
C06771=1206.323,-7.725,-42.548,-179.788,5.547,148.911
C06772=1206.318,-7.475,-42.562,-179.785,5.548,148.910
C06773=1206.313,-7.226,-42.575,-179.782,5.548,148.909
C06774=1206.308,-6.976,-42.589,-179.781,5.548,148.909
C06775=1206.303,-6.726,-42.603,-179.778,5.549,148.908
C06776=1206.297,-6.476,-42.616,-179.776,5.549,148.907
C06777=1206.293,-6.227,-42.630,-179.773,5.550,148.907
C06778=1206.287,-5.978,-42.644,-179.770,5.550,148.906
C06779=1206.282,-5.728,-42.658,-179.768,5.550,148.905
C06780=1206.277,-5.478,-42.672,-179.765,5.550,148.905
C06781=1206.272,-5.229,-42.685,-179.763,5.551,148.904
C06782=1206.267,-4.980,-42.699,-179.761,5.552,148.904
C06783=1206.262,-4.730,-42.714,-179.758,5.552,148.903
C06784=1206.256,-4.480,-42.727,-179.755,5.553,148.902
C06785=1206.251,-4.231,-42.741,-179.753,5.552,148.901
C06786=1206.247,-3.981,-42.755,-179.751,5.553,148.901
C06787=1206.242,-3.732,-42.769,-179.748,5.553,148.900
C06788=1206.236,-3.482,-42.782,-179.745,5.554,148.899
C06789=1206.231,-3.232,-42.797,-179.743,5.554,148.899
C06790=1206.226,-2.983,-42.810,-179.741,5.555,148.898
C06791=1206.222,-2.734,-42.824,-179.738,5.555,148.898
C06792=1206.217,-2.484,-42.838,-179.736,5.556,148.897
C06793=1206.211,-2.234,-42.852,-179.733,5.556,148.896
C06794=1206.206,-1.985,-42.866,-179.730,5.557,148.895
C06795=1206.201,-1.735,-42.880,-179.728,5.557,148.895
C06796=1206.196,-1.485,-42.894,-179.725,5.558,148.894
C06797=1206.191,-1.237,-42.908,-179.724,5.558,148.894
C06798=1206.186,-0.987,-42.922,-179.721,5.558,148.893
C06799=1206.181,-0.737,-42.936,-179.718,5.559,148.892
C06800=1206.176,-0.487,-42.950,-179.716,5.559,148.892
C06801=1206.170,-0.238,-42.964,-179.713,5.560,148.891
C06802=1206.165,0.012,-42.978,-179.710,5.560,148.890
C06803=1206.160,0.262,-42.992,-179.708,5.560,148.890
C06804=1206.155,0.511,-43.007,-179.706,5.560,148.889
C06805=1206.150,0.760,-43.021,-179.703,5.561,148.888
C06806=1206.146,1.010,-43.034,-179.701,5.562,148.888
C06807=1206.141,1.259,-43.049,-179.698,5.562,148.887
C06808=1206.136,1.509,-43.063,-179.695,5.563,148.886
C06809=1206.130,1.758,-43.077,-179.693,5.563,148.886
C06810=1206.125,2.008,-43.091,-179.691,5.563,148.885
C06811=1206.120,2.258,-43.105,-179.688,5.563,148.884
C06812=1206.115,2.507,-43.120,-179.686,5.564,148.884
C06813=1206.109,2.776,-43.134,-179.683,5.564,148.883
C06814=1206.104,3.045,-43.149,-179.680,5.565,148.882
C06815=1206.099,3.314,-43.165,-179.677,5.565,148.881
C06816=1206.093,3.584,-43.180,-179.675,5.566,148.881
C06817=1206.088,3.833,-43.194,-179.672,5.566,148.880
C06818=1206.083,4.083,-43.208,-179.670,5.567,148.880
C06819=1206.078,4.332,-43.222,-179.667,5.568,148.879
C06820=1206.073,4.582,-43.237,-179.665,5.568,148.878
C06821=1206.068,4.832,-43.251,-179.663,5.568,148.878
C06822=1206.063,5.081,-43.266,-179.660,5.568,148.877
C06823=1206.058,5.330,-43.280,-179.657,5.569,148.876
C06824=1206.053,5.579,-43.294,-179.655,5.569,148.876
C06825=1206.048,5.829,-43.308,-179.653,5.570,148.875
C06826=1206.043,6.079,-43.323,-179.650,5.571,148.874
C06827=1206.038,6.328,-43.337,-179.647,5.571,148.874
C06828=1206.033,6.578,-43.351,-179.645,5.571,148.873
C06829=1206.028,6.828,-43.365,-179.642,5.571,148.872
C06830=1206.022,7.077,-43.379,-179.640,5.572,148.872
C06831=1206.018,7.327,-43.394,-179.637,5.573,148.871
C06832=1206.012,7.576,-43.409,-179.635,5.573,148.870
C06833=1206.007,7.826,-43.423,-179.632,5.574,148.870
C06834=1206.002,8.075,-43.438,-179.630,5.574,148.869
C06835=1205.997,8.325,-43.452,-179.627,5.575,148.868
C06836=1205.992,8.575,-43.466,-179.625,5.575,148.868
C06837=1205.987,8.824,-43.480,-179.622,5.575,148.867
C06838=1205.982,9.073,-43.495,-179.620,5.576,148.866
C06839=1205.977,9.323,-43.509,-179.618,5.576,148.866
C06840=1205.972,9.572,-43.524,-179.615,5.577,148.865
C06841=1205.967,9.822,-43.538,-179.612,5.577,148.865
C06842=1205.962,10.072,-43.552,-179.610,5.578,148.864
C06843=1205.957,10.321,-43.568,-179.607,5.579,148.863
C06844=1205.952,10.571,-43.582,-179.604,5.579,148.862
C06845=1205.946,10.820,-43.596,-179.602,5.579,148.862
C06846=1205.941,11.070,-43.610,-179.600,5.580,148.861
C06847=1205.937,11.319,-43.625,-179.597,5.580,148.861
C06848=1205.932,11.568,-43.640,-179.595,5.581,148.860
C06849=1205.927,11.818,-43.654,-179.592,5.581,148.859
C06850=1205.921,12.068,-43.669,-179.589,5.582,148.859
C06851=1205.917,12.317,-43.684,-179.587,5.582,148.858
C06852=1205.912,12.567,-43.698,-179.585,5.583,148.857
C06853=1205.907,12.817,-43.712,-179.582,5.584,148.857
C06854=1205.902,13.066,-43.727,-179.579,5.584,148.856
C06855=1205.897,13.315,-43.742,-179.577,5.584,148.855
C06856=1205.891,13.565,-43.756,-179.575,5.584,148.855
C06857=1205.887,13.815,-43.771,-179.572,5.585,148.854
C06858=1205.881,14.064,-43.785,-179.570,5.586,148.854
C06859=1205.876,14.313,-43.800,-179.567,5.586,148.853
C06860=1205.872,14.562,-43.815,-179.565,5.587,148.852
C06861=1205.866,14.812,-43.830,-179.562,5.587,148.852
C06862=1205.861,15.061,-43.845,-179.559,5.588,148.851
C06863=1205.856,15.311,-43.859,-179.557,5.588,148.850
C06864=1205.851,15.561,-43.873,-179.554,5.589,148.849
C06865=1205.846,15.810,-43.889,-179.552,5.590,148.849
C06866=1205.841,16.060,-43.903,-179.550,5.589,148.848
C06867=1205.836,16.309,-43.918,-179.547,5.590,148.848
C06868=1205.831,16.559,-43.932,-179.544,5.590,148.847
C06869=1205.826,16.809,-43.947,-179.542,5.591,148.846
C06870=1205.821,17.058,-43.962,-179.539,5.591,148.846
C06871=1205.816,17.308,-43.976,-179.537,5.592,148.845
C06872=1205.811,17.557,-43.992,-179.534,5.593,148.844
C06873=1205.806,17.807,-44.006,-179.532,5.593,148.844
C06874=1205.801,18.056,-44.021,-179.529,5.594,148.843
C06875=1205.796,18.306,-44.035,-179.526,5.594,148.842
C06876=1205.791,18.555,-44.051,-179.524,5.595,148.842
C06877=1205.786,18.805,-44.065,-179.522,5.596,148.841
C06878=1205.781,19.054,-44.080,-179.519,5.596,148.841
C06879=1205.775,19.304,-44.095,-179.517,5.596,148.840
C06880=1205.771,19.553,-44.110,-179.514,5.596,148.839
C06881=1205.766,19.803,-44.124,-179.512,5.597,148.839
C06882=1205.760,20.052,-44.140,-179.509,5.597,148.838
C06883=1205.755,20.302,-44.154,-179.507,5.598,148.837
C06884=1205.751,20.551,-44.169,-179.504,5.599,148.837
C06885=1205.745,20.800,-44.185,-179.501,5.599,148.836
C06886=1205.741,21.051,-44.200,-179.499,5.600,148.835
C06887=1205.736,21.300,-44.215,-179.496,5.600,148.835
C06888=1205.731,21.550,-44.229,-179.493,5.601,148.834
C06889=1205.726,21.799,-44.244,-179.491,5.602,148.834
C06890=1205.721,22.048,-44.260,-179.489,5.602,148.833
C06891=1205.716,22.298,-44.274,-179.486,5.603,148.832
C06892=1205.711,22.547,-44.289,-179.483,5.603,148.832
C06893=1205.705,22.797,-44.304,-179.481,5.604,148.831
C06894=1205.701,23.046,-44.319,-179.479,5.605,148.830
C06895=1205.695,23.296,-44.335,-179.477,5.604,148.830
C06896=1205.690,23.545,-44.349,-179.474,5.605,148.829
C06897=1205.685,23.795,-44.365,-179.471,5.605,148.828
C06898=1205.680,24.044,-44.380,-179.469,5.606,148.828
C06899=1205.676,24.294,-44.394,-179.466,5.607,148.827
C06900=1205.671,24.544,-44.410,-179.464,5.607,148.827
C06901=1205.666,24.793,-44.425,-179.461,5.608,148.826
C06902=1205.661,25.042,-44.440,-179.458,5.608,148.825
C06903=1205.656,25.292,-44.455,-179.456,5.609,148.825
C06904=1205.650,25.541,-44.470,-179.453,5.609,148.824
C06905=1205.646,25.790,-44.485,-179.451,5.610,148.823
C06906=1205.640,26.040,-44.500,-179.448,5.611,148.823
C06907=1205.636,26.290,-44.516,-179.446,5.611,148.822
C06908=1205.630,26.539,-44.531,-179.443,5.612,148.821
C06909=1205.626,26.789,-44.546,-179.440,5.612,148.821
C06910=1205.620,27.039,-44.561,-179.438,5.613,148.820
C06911=1205.615,27.288,-44.576,-179.436,5.614,148.820
C06912=1205.610,27.537,-44.592,-179.433,5.614,148.819
C06913=1205.605,27.786,-44.607,-179.430,5.615,148.818
C06914=1205.601,28.036,-44.622,-179.428,5.615,148.818
C06915=1205.596,28.285,-44.637,-179.425,5.616,148.817
C06916=1205.590,28.535,-44.652,-179.423,5.617,148.816
C06917=1205.585,28.804,-44.669,-179.420,5.617,148.816
C06918=1205.580,29.073,-44.685,-179.418,5.618,148.815
C06919=1205.574,29.341,-44.702,-179.415,5.618,148.814
C06920=1205.569,29.610,-44.718,-179.412,5.619,148.813
C06921=1205.564,29.859,-44.733,-179.410,5.619,148.813
C06922=1205.559,30.109,-44.749,-179.407,5.620,148.812
C06923=1205.554,30.359,-44.764,-179.404,5.620,148.812
C06924=1205.549,30.608,-44.780,-179.402,5.621,148.811
C06925=1205.544,30.857,-44.795,-179.399,5.622,148.810
C06926=1205.539,31.106,-44.811,-179.397,5.622,148.810
C06927=1205.534,31.357,-44.826,-179.394,5.623,148.809
C06928=1205.529,31.606,-44.841,-179.392,5.623,148.808
C06929=1205.524,31.856,-44.856,-179.389,5.624,148.808
C06930=1205.519,32.105,-44.871,-179.386,5.625,148.807
C06931=1205.514,32.354,-44.887,-179.384,5.625,148.807
C06932=1205.509,32.604,-44.903,-179.382,5.626,148.806
C06933=1205.504,32.853,-44.918,-179.379,5.626,148.805
C06934=1205.499,33.103,-44.933,-179.376,5.627,148.805
C06935=1205.493,33.352,-44.949,-179.374,5.628,148.804
C06936=1205.489,33.602,-44.964,-179.371,5.628,148.804
C06937=1205.484,33.851,-44.980,-179.369,5.629,148.803
C06938=1205.478,34.101,-44.996,-179.366,5.629,148.802
C06939=1205.474,34.350,-45.011,-179.364,5.630,148.802
C06940=1205.469,34.600,-45.027,-179.361,5.631,148.801
C06941=1205.464,34.849,-45.042,-179.359,5.631,148.800
C06942=1205.459,35.098,-45.057,-179.356,5.632,148.800
C06943=1205.454,35.347,-45.073,-179.353,5.632,148.799
C06944=1205.449,35.597,-45.089,-179.351,5.633,148.798
C06945=1205.445,35.846,-45.104,-179.349,5.634,148.798
C06946=1205.439,36.096,-45.120,-179.346,5.634,148.797
C06947=1205.434,36.346,-45.136,-179.343,5.635,148.797
C06948=1205.429,36.595,-45.151,-179.341,5.635,148.796
C06949=1205.424,36.844,-45.166,-179.338,5.636,148.795
C06950=1205.419,37.094,-45.182,-179.336,5.637,148.795
C06951=1205.414,37.344,-45.198,-179.333,5.637,148.794
C06952=1205.409,37.593,-45.214,-179.331,5.638,148.793
C06953=1205.404,37.842,-45.229,-179.328,5.639,148.793
C06954=1205.400,38.092,-45.245,-179.325,5.639,148.792
C06955=1205.394,38.341,-45.261,-179.323,5.640,148.792
C06956=1205.389,38.591,-45.276,-179.321,5.640,148.791
C06957=1205.384,38.841,-45.292,-179.318,5.641,148.790
C06958=1205.379,39.090,-45.307,-179.315,5.642,148.790
C06959=1205.374,39.339,-45.324,-179.313,5.642,148.789
C06960=1205.370,39.589,-45.340,-179.311,5.643,148.788
C06961=1205.364,39.838,-45.355,-179.308,5.643,148.788
C06962=1205.359,40.088,-45.371,-179.305,5.644,148.787
C06963=1205.355,40.337,-45.386,-179.303,5.645,148.786
C06964=1205.350,40.586,-45.402,-179.300,5.645,148.786
C06965=1205.344,40.836,-45.418,-179.297,5.647,148.785
C06966=1205.339,41.086,-45.434,-179.295,5.647,148.785
C06967=1205.334,41.335,-45.450,-179.292,5.648,148.784
C06968=1205.329,41.584,-45.466,-179.290,5.649,148.784
C06969=1205.325,41.834,-45.481,-179.287,5.649,148.783
C06970=1205.320,42.083,-45.497,-179.285,5.650,148.782
C06971=1205.315,42.333,-45.513,-179.282,5.650,148.782
C06972=1205.310,42.582,-45.529,-179.279,5.651,148.781
C06973=1205.304,42.831,-45.545,-179.277,5.652,148.780
C06974=1205.300,43.081,-45.561,-179.274,5.652,148.780
C06975=1205.294,43.330,-45.577,-179.272,5.653,148.779
C06976=1205.289,43.580,-45.593,-179.269,5.653,148.778
C06977=1205.284,43.830,-45.608,-179.267,5.654,148.778
C06978=1205.280,44.078,-45.624,-179.264,5.655,148.777
C06979=1205.275,44.328,-45.640,-179.262,5.655,148.777
C06980=1205.270,44.577,-45.656,-179.259,5.656,148.776
C06981=1205.265,44.827,-45.672,-179.257,5.657,148.776
C06982=1205.260,45.077,-45.688,-179.254,5.657,148.775
C06983=1205.255,45.325,-45.704,-179.252,5.658,148.774
C06984=1205.250,45.575,-45.720,-179.249,5.658,148.773
C06985=1205.245,45.824,-45.737,-179.247,5.659,148.773
C06986=1205.240,46.074,-45.753,-179.244,5.661,148.772
C06987=1205.235,46.324,-45.768,-179.241,5.661,148.772
C06988=1205.230,46.573,-45.785,-179.238,5.662,148.771
C06989=1205.225,46.823,-45.800,-179.236,5.662,148.770
C06990=1205.220,47.072,-45.817,-179.234,5.663,148.770
C06991=1205.215,47.322,-45.833,-179.231,5.664,148.769
C06992=1205.210,47.570,-45.849,-179.228,5.664,148.769
C06993=1205.205,47.820,-45.865,-179.226,5.665,148.768
C06994=1205.200,48.069,-45.881,-179.224,5.666,148.767
C06995=1205.195,48.319,-45.897,-179.221,5.666,148.767
C06996=1205.190,48.568,-45.913,-179.218,5.667,148.766
C06997=1205.185,48.818,-45.929,-179.216,5.667,148.765
C06998=1205.180,49.067,-45.946,-179.213,5.668,148.765
C06999=1205.176,49.317,-45.962,-179.211,5.669,148.764
C07000=1205.170,49.566,-45.978,-179.208,5.670,148.764
C07001=1205.166,49.816,-45.994,-179.205,5.671,148.763
C07002=1205.161,50.065,-46.010,-179.203,5.672,148.763
C07003=1205.156,50.315,-46.026,-179.200,5.672,148.762
C07004=1205.151,50.564,-46.042,-179.198,5.673,148.761
C07005=1205.146,50.813,-46.059,-179.195,5.673,148.761
C07006=1205.141,51.063,-46.075,-179.193,5.674,148.760
C07007=1205.136,51.312,-46.091,-179.190,5.675,148.759
C07008=1205.130,51.562,-46.108,-179.188,5.675,148.759
C07009=1205.126,51.811,-46.124,-179.185,5.676,148.758
C07010=1205.121,52.061,-46.141,-179.183,5.677,148.758
C07011=1205.116,52.310,-46.156,-179.180,5.677,148.757
C07012=1205.111,52.560,-46.173,-179.177,5.679,148.756
C07013=1205.106,52.808,-46.189,-179.175,5.679,148.756
C07014=1205.102,53.058,-46.205,-179.172,5.680,148.755
C07015=1205.096,53.307,-46.222,-179.169,5.681,148.755
C07016=1205.092,53.557,-46.238,-179.167,5.681,148.754
C07017=1205.086,53.806,-46.255,-179.165,5.682,148.753
C07018=1205.081,54.056,-46.271,-179.162,5.682,148.753
C07019=1205.076,54.305,-46.288,-179.159,5.683,148.752
C07020=1205.072,54.555,-46.304,-179.157,5.684,148.751
C07021=1205.066,54.823,-46.321,-179.154,5.685,148.751
C07022=1205.061,55.092,-46.340,-179.151,5.686,148.750
C07023=1205.055,55.360,-46.357,-179.149,5.686,148.750
C07024=1205.051,55.629,-46.375,-179.146,5.687,148.749
C07025=1205.045,55.878,-46.391,-179.143,5.688,148.748
C07026=1205.041,56.127,-46.407,-179.140,5.689,148.748
C07027=1205.035,56.377,-46.424,-179.138,5.689,148.747
C07028=1205.031,56.626,-46.441,-179.136,5.690,148.747
C07029=1205.026,56.876,-46.458,-179.133,5.691,148.746
C07030=1205.021,57.125,-46.473,-179.130,5.691,148.745
C07031=1205.015,57.375,-46.490,-179.128,5.692,148.745
C07032=1205.010,57.623,-46.507,-179.125,5.693,148.744
C07033=1205.006,57.873,-46.523,-179.122,5.694,148.744
C07034=1205.001,58.122,-46.540,-179.120,5.695,148.743
C07035=1204.996,58.372,-46.557,-179.117,5.696,148.742
C07036=1204.991,58.622,-46.573,-179.115,5.696,148.742
C07037=1204.986,58.871,-46.590,-179.112,5.697,148.741
C07038=1204.981,59.120,-46.606,-179.110,5.698,148.741
C07039=1204.976,59.370,-46.623,-179.107,5.698,148.740
C07040=1204.972,59.619,-46.640,-179.105,5.699,148.739
C07041=1204.966,59.868,-46.656,-179.102,5.700,148.739
C07042=1204.961,60.118,-46.673,-179.099,5.701,148.738
C07043=1204.957,60.367,-46.690,-179.097,5.702,148.738
C07044=1204.952,60.616,-46.706,-179.094,5.702,148.737
C07045=1204.946,60.866,-46.724,-179.092,5.703,148.736
C07046=1204.942,61.116,-46.740,-179.089,5.704,148.736
C07047=1204.937,61.365,-46.756,-179.087,5.704,148.735
C07048=1204.931,61.615,-46.773,-179.084,5.706,148.734
C07049=1204.927,61.864,-46.790,-179.081,5.706,148.734
C07050=1204.922,62.113,-46.806,-179.079,5.707,148.733
C07051=1204.917,62.363,-46.823,-179.076,5.708,148.733
C07052=1204.912,62.612,-46.840,-179.074,5.708,148.732
C07053=1204.907,62.861,-46.856,-179.071,5.709,148.732
C07054=1204.902,63.111,-46.874,-179.069,5.710,148.731
C07055=1204.897,63.360,-46.890,-179.066,5.711,148.730
C07056=1204.893,63.610,-46.907,-179.063,5.712,148.730
C07057=1204.887,63.859,-46.924,-179.061,5.712,148.729
C07058=1204.883,64.108,-46.941,-179.058,5.713,148.729
C07059=1204.878,64.357,-46.958,-179.056,5.714,148.728
C07060=1204.873,64.607,-46.975,-179.053,5.714,148.727
C07061=1204.868,64.856,-46.991,-179.050,5.716,148.727
C07062=1204.863,65.105,-47.009,-179.048,5.717,148.726
C07063=1204.858,65.355,-47.025,-179.045,5.717,148.726
C07064=1204.853,65.604,-47.042,-179.043,5.718,148.725
C07065=1204.848,65.853,-47.059,-179.041,5.719,148.725
C07066=1204.843,66.103,-47.076,-179.038,5.719,148.724
C07067=1204.838,66.353,-47.093,-179.035,5.720,148.723
C07068=1204.833,66.602,-47.111,-179.033,5.722,148.723
C07069=1204.828,66.851,-47.127,-179.030,5.722,148.722
C07070=1204.823,67.101,-47.144,-179.027,5.723,148.721
C07071=1204.819,67.350,-47.161,-179.025,5.723,148.721
C07072=1204.814,67.600,-47.178,-179.023,5.724,148.720
C07073=1204.808,67.849,-47.195,-179.019,5.725,148.720
C07074=1204.804,68.097,-47.212,-179.017,5.726,148.719
C07075=1204.799,68.347,-47.229,-179.015,5.727,148.719
C07076=1204.795,68.597,-47.246,-179.012,5.727,148.718
C07077=1204.789,68.847,-47.263,-179.009,5.728,148.717
C07078=1204.784,69.095,-47.280,-179.007,5.729,148.717
C07079=1204.779,69.344,-47.298,-179.004,5.730,148.716
C07080=1204.774,69.594,-47.315,-179.001,5.731,148.716
C07081=1204.770,69.844,-47.331,-178.999,5.732,148.715
C07082=1204.765,70.093,-47.349,-178.997,5.732,148.714
C07083=1204.760,70.342,-47.366,-178.994,5.733,148.714
C07084=1204.754,70.592,-47.383,-178.991,5.735,148.713
C07085=1204.750,70.841,-47.400,-178.989,5.735,148.713
C07086=1204.745,71.090,-47.418,-178.986,5.736,148.712
C07087=1204.741,71.340,-47.434,-178.984,5.737,148.712
C07088=1204.735,71.589,-47.452,-178.981,5.737,148.711
C07089=1204.730,71.839,-47.470,-178.978,5.739,148.710
C07090=1204.725,72.087,-47.486,-178.976,5.740,148.710
C07091=1204.720,72.337,-47.503,-178.973,5.740,148.709
C07092=1204.716,72.586,-47.521,-178.971,5.741,148.709
C07093=1204.711,72.836,-47.538,-178.968,5.742,148.708
C07094=1204.706,73.086,-47.555,-178.965,5.743,148.707
C07095=1204.701,73.335,-47.572,-178.963,5.744,148.707
C07096=1204.696,73.584,-47.590,-178.961,5.744,148.706
C07097=1204.691,73.834,-47.608,-178.958,5.745,148.706
C07098=1204.686,74.082,-47.624,-178.955,5.746,148.705
C07099=1204.681,74.332,-47.641,-178.953,5.747,148.705
C07100=1204.676,74.581,-47.659,-178.950,5.748,148.704
C07101=1204.672,74.831,-47.676,-178.947,5.748,148.703
C07102=1204.667,75.080,-47.694,-178.945,5.749,148.703
C07103=1204.661,75.330,-47.711,-178.943,5.750,148.702
C07104=1204.657,75.579,-47.729,-178.939,5.751,148.702
C07105=1204.652,75.828,-47.746,-178.937,5.752,148.701
C07106=1204.647,76.078,-47.764,-178.935,5.753,148.701
C07107=1204.643,76.327,-47.780,-178.932,5.754,148.700
C07108=1204.638,76.576,-47.798,-178.929,5.755,148.699
C07109=1204.632,76.825,-47.815,-178.927,5.756,148.699
C07110=1204.628,77.074,-47.833,-178.924,5.757,148.698
C07111=1204.622,77.324,-47.850,-178.922,5.757,148.698
C07112=1204.618,77.573,-47.868,-178.919,5.758,148.697
C07113=1204.612,77.823,-47.885,-178.916,5.759,148.697
C07114=1204.608,78.072,-47.903,-178.914,5.760,148.696
C07115=1204.603,78.322,-47.920,-178.911,5.761,148.695
C07116=1204.598,78.571,-47.938,-178.909,5.761,148.695
C07117=1204.593,78.820,-47.956,-178.906,5.763,148.694
C07118=1204.588,79.070,-47.973,-178.903,5.763,148.694
C07119=1204.584,79.319,-47.990,-178.901,5.764,148.693
C07120=1204.579,79.568,-48.008,-178.898,5.765,148.692
C07121=1204.574,79.818,-48.026,-178.896,5.767,148.692
C07122=1204.569,80.067,-48.044,-178.893,5.767,148.691
C07123=1204.564,80.316,-48.060,-178.891,5.768,148.691
C07124=1204.559,80.565,-48.078,-178.888,5.769,148.690
C07125=1204.554,80.834,-48.097,-178.885,5.770,148.690
C07126=1204.549,81.103,-48.116,-178.883,5.771,148.689
C07127=1204.543,81.370,-48.136,-178.879,5.772,148.688
C07128=1204.538,81.639,-48.154,-178.877,5.773,148.688
C07129=1204.533,81.888,-48.172,-178.875,5.773,148.687
C07130=1204.528,82.137,-48.190,-178.871,5.775,148.687
C07131=1204.523,82.387,-48.207,-178.869,5.776,148.686
C07132=1204.519,82.636,-48.225,-178.867,5.776,148.686
C07133=1204.514,82.885,-48.243,-178.864,5.777,148.685
C07134=1204.508,83.135,-48.260,-178.861,5.779,148.684
C07135=1204.504,83.384,-48.278,-178.859,5.779,148.684
C07136=1204.499,83.633,-48.296,-178.856,5.780,148.683
C07137=1204.494,83.883,-48.314,-178.854,5.781,148.683
C07138=1204.489,84.133,-48.332,-178.851,5.782,148.682
C07139=1204.484,84.382,-48.350,-178.849,5.783,148.682
C07140=1204.479,84.631,-48.368,-178.846,5.784,148.681
C07141=1204.475,84.880,-48.385,-178.843,5.785,148.680
C07142=1204.470,85.129,-48.403,-178.841,5.786,148.680
C07143=1204.465,85.379,-48.420,-178.838,5.787,148.679
C07144=1204.460,85.628,-48.438,-178.836,5.787,148.679
C07145=1204.455,85.878,-48.456,-178.833,5.789,148.678
C07146=1204.450,86.127,-48.474,-178.830,5.789,148.678
C07147=1204.445,86.376,-48.492,-178.828,5.790,148.677
C07148=1204.440,86.625,-48.510,-178.825,5.791,148.676
C07149=1204.435,86.874,-48.528,-178.823,5.793,148.676
C07150=1204.431,87.124,-48.546,-178.820,5.793,148.675
C07151=1204.426,87.374,-48.564,-178.817,5.794,148.675
C07152=1204.421,87.623,-48.582,-178.815,5.796,148.674
C07153=1204.416,87.872,-48.600,-178.812,5.796,148.674
C07154=1204.411,88.121,-48.618,-178.810,5.797,148.673
C07155=1204.406,88.371,-48.636,-178.807,5.798,148.673
C07156=1204.401,88.620,-48.654,-178.804,5.799,148.672
C07157=1204.396,88.869,-48.672,-178.802,5.800,148.672
C07158=1204.392,89.118,-48.690,-178.799,5.800,148.671
C07159=1204.387,89.368,-48.708,-178.797,5.802,148.671
C07160=1204.382,89.617,-48.726,-178.794,5.803,148.670
C07161=1204.377,89.866,-48.744,-178.791,5.803,148.669
C07162=1204.373,90.116,-48.762,-178.789,5.805,148.669
C07163=1204.368,90.365,-48.780,-178.786,5.806,148.668
C07164=1204.363,90.614,-48.798,-178.784,5.807,148.668
C07165=1204.358,90.864,-48.816,-178.781,5.807,148.667
C07166=1204.353,91.113,-48.835,-178.779,5.809,148.667
C07167=1204.348,91.362,-48.853,-178.776,5.810,148.666
C07168=1204.343,91.612,-48.871,-178.773,5.810,148.665
C07169=1204.338,91.861,-48.889,-178.771,5.812,148.665
C07170=1204.333,92.110,-48.907,-178.768,5.812,148.664
C07171=1204.329,92.360,-48.925,-178.766,5.813,148.664
C07172=1204.324,92.609,-48.943,-178.763,5.815,148.663
C07173=1204.319,92.858,-48.961,-178.761,5.816,148.663
C07174=1204.314,93.107,-48.980,-178.758,5.816,148.662
C07175=1204.309,93.356,-48.998,-178.755,5.818,148.662
C07176=1204.304,93.606,-49.017,-178.753,5.819,148.661
C07177=1204.299,93.855,-49.035,-178.750,5.819,148.660
C07178=1204.295,94.104,-49.053,-178.747,5.821,148.660
C07179=1204.290,94.354,-49.070,-178.745,5.821,148.659
C07180=1204.285,94.603,-49.088,-178.743,5.822,148.659
C07181=1204.280,94.852,-49.108,-178.739,5.824,148.658
C07182=1204.275,95.102,-49.126,-178.737,5.824,148.658
C07183=1204.270,95.351,-49.144,-178.735,5.825,148.657
C07184=1204.265,95.600,-49.162,-178.731,5.827,148.657
C07185=1204.261,95.850,-49.180,-178.729,5.828,148.656
C07186=1204.256,96.099,-49.200,-178.727,5.828,148.656
C07187=1204.251,96.348,-49.218,-178.724,5.830,148.655
C07188=1204.246,96.597,-49.236,-178.721,5.831,148.654
C07189=1204.241,96.847,-49.254,-178.719,5.831,148.654
C07190=1204.237,97.095,-49.273,-178.716,5.833,148.653
C07191=1204.231,97.345,-49.291,-178.713,5.833,148.653
C07192=1204.226,97.594,-49.309,-178.711,5.834,148.652
C07193=1204.222,97.844,-49.328,-178.708,5.836,148.652
C07194=1204.217,98.093,-49.346,-178.706,5.837,148.651
C07195=1204.212,98.342,-49.365,-178.703,5.837,148.651
C07196=1204.207,98.592,-49.383,-178.701,5.839,148.650
C07197=1204.203,98.840,-49.402,-178.698,5.840,148.650
C07198=1204.197,99.090,-49.420,-178.696,5.841,148.649
C07199=1204.193,99.340,-49.439,-178.693,5.842,148.649
C07200=1204.188,99.588,-49.458,-178.691,5.843,148.648
C07201=1204.183,99.838,-49.476,-178.688,5.843,148.647
C07202=1204.178,100.087,-49.494,-178.685,5.845,148.647
C07203=1204.174,100.336,-49.513,-178.683,5.846,148.646
C07204=1204.169,100.585,-49.531,-178.679,5.847,148.646
C07205=1204.163,100.834,-49.550,-178.677,5.848,148.645
C07206=1204.159,101.084,-49.569,-178.675,5.849,148.645
C07207=1204.154,101.333,-49.587,-178.672,5.850,148.644
C07208=1204.149,101.582,-49.606,-178.669,5.851,148.644
C07209=1204.145,101.832,-49.624,-178.667,5.852,148.643
C07210=1204.140,102.081,-49.643,-178.664,5.853,148.643
C07211=1204.135,102.331,-49.662,-178.662,5.854,148.642
C07212=1204.130,102.579,-49.681,-178.659,5.856,148.642
C07213=1204.125,102.829,-49.699,-178.657,5.857,148.641
C07214=1204.121,103.078,-49.718,-178.654,5.857,148.640
C07215=1204.116,103.327,-49.736,-178.651,5.859,148.640
C07216=1204.110,103.576,-49.756,-178.649,5.860,148.639
C07217=1204.106,103.826,-49.774,-178.647,5.861,148.639
C07218=1204.101,104.075,-49.793,-178.643,5.862,148.638
C07219=1204.096,104.324,-49.811,-178.641,5.863,148.638
C07220=1204.092,104.573,-49.830,-178.638,5.864,148.637
C07221=1204.086,104.823,-49.849,-178.636,5.865,148.637
C07222=1204.082,105.072,-49.868,-178.633,5.866,148.636
C07223=1204.076,105.322,-49.887,-178.630,5.867,148.636
C07224=1204.072,105.570,-49.905,-178.628,5.868,148.635
C07225=1204.067,105.820,-49.925,-178.625,5.870,148.635
C07226=1204.062,106.069,-49.943,-178.623,5.871,148.634
C07227=1204.057,106.318,-49.963,-178.620,5.871,148.634
C07228=1204.053,106.568,-49.980,-178.617,5.873,148.633
C07229=1204.048,106.836,-50.002,-178.615,5.873,148.632
C07230=1204.042,107.105,-50.022,-178.612,5.875,148.632
C07231=1204.037,107.372,-50.042,-178.609,5.877,148.631
C07232=1204.032,107.641,-50.063,-178.606,5.877,148.631
C07233=1204.027,107.890,-50.081,-178.604,5.879,148.630
C07234=1204.022,108.140,-50.100,-178.601,5.880,148.630
C07235=1204.017,108.389,-50.120,-178.599,5.880,148.629
C07236=1204.013,108.639,-50.138,-178.596,5.882,148.629
C07237=1204.007,108.887,-50.157,-178.593,5.883,148.628
C07238=1204.003,109.136,-50.176,-178.590,5.884,148.628
C07239=1203.998,109.386,-50.195,-178.588,5.885,148.627
C07240=1203.993,109.635,-50.214,-178.586,5.886,148.627
C07241=1203.988,109.884,-50.233,-178.583,5.888,148.626
C07242=1203.984,110.133,-50.252,-178.580,5.888,148.626
C07243=1203.979,110.383,-50.271,-178.578,5.890,148.625
C07244=1203.973,110.632,-50.290,-178.575,5.890,148.625
C07245=1203.969,110.881,-50.309,-178.572,5.892,148.624
C07246=1203.964,111.130,-50.329,-178.570,5.893,148.623
C07247=1203.960,111.379,-50.348,-178.567,5.894,148.623
C07248=1203.954,111.629,-50.366,-178.564,5.895,148.622
C07249=1203.950,111.878,-50.386,-178.562,5.896,148.622
C07250=1203.945,112.127,-50.405,-178.559,5.898,148.621
C07251=1203.940,112.377,-50.424,-178.557,5.898,148.621
C07252=1203.935,112.625,-50.444,-178.554,5.900,148.620
C07253=1203.931,112.875,-50.463,-178.552,5.901,148.620
C07254=1203.926,113.125,-50.482,-178.549,5.902,148.620
C07255=1203.921,113.374,-50.501,-178.546,5.903,148.619
C07256=1203.917,113.623,-50.520,-178.544,5.904,148.619
C07257=1203.911,113.872,-50.539,-178.541,5.906,148.618
C07258=1203.907,114.121,-50.559,-178.539,5.906,148.617
C07259=1203.902,114.370,-50.578,-178.536,5.908,148.617
C07260=1203.897,114.620,-50.597,-178.534,5.909,148.616
C07261=1203.892,114.868,-50.616,-178.530,5.910,148.616
C07262=1203.888,115.118,-50.636,-178.528,5.911,148.615
C07263=1203.883,115.367,-50.655,-178.526,5.912,148.615
C07264=1203.878,115.616,-50.674,-178.523,5.914,148.614
C07265=1203.873,115.866,-50.694,-178.520,5.914,148.614
C07266=1203.868,116.114,-50.713,-178.518,5.916,148.613
C07267=1203.864,116.364,-50.733,-178.515,5.917,148.613
C07268=1203.858,116.613,-50.752,-178.512,5.918,148.612
C07269=1203.854,116.862,-50.771,-178.510,5.919,148.612
C07270=1203.850,117.111,-50.791,-178.507,5.921,148.611
C07271=1203.844,117.360,-50.810,-178.505,5.922,148.611
C07272=1203.839,117.610,-50.829,-178.502,5.923,148.610
C07273=1203.834,117.859,-50.849,-178.500,5.924,148.610
C07274=1203.830,118.108,-50.868,-178.496,5.925,148.609
C07275=1203.825,118.358,-50.887,-178.494,5.926,148.609
C07276=1203.820,118.606,-50.907,-178.492,5.928,148.608
C07277=1203.815,118.856,-50.926,-178.489,5.929,148.608
C07278=1203.811,119.106,-50.946,-178.487,5.930,148.607
C07279=1203.806,119.354,-50.965,-178.484,5.931,148.607
C07280=1203.801,119.604,-50.984,-178.482,5.932,148.606
C07281=1203.797,119.853,-51.005,-178.478,5.933,148.606
C07282=1203.791,120.102,-51.024,-178.476,5.934,148.605
C07283=1203.787,120.351,-51.044,-178.474,5.936,148.605
C07284=1203.782,120.601,-51.063,-178.471,5.937,148.604
C07285=1203.777,120.850,-51.083,-178.468,5.938,148.604
C07286=1203.773,121.099,-51.102,-178.466,5.939,148.603
C07287=1203.768,121.348,-51.122,-178.463,5.941,148.603
C07288=1203.763,121.597,-51.141,-178.460,5.941,148.602
C07289=1203.758,121.846,-51.161,-178.458,5.943,148.602
C07290=1203.753,122.096,-51.181,-178.456,5.944,148.601
C07291=1203.748,122.345,-51.200,-178.452,5.946,148.601
C07292=1203.744,122.594,-51.220,-178.450,5.947,148.600
C07293=1203.739,122.843,-51.240,-178.447,5.948,148.600
C07294=1203.733,123.092,-51.259,-178.445,5.949,148.599
C07295=1203.729,123.342,-51.279,-178.442,5.951,148.599
C07296=1203.725,123.590,-51.299,-178.440,5.951,148.598
C07297=1203.720,123.840,-51.318,-178.437,5.953,148.598
C07298=1203.715,124.089,-51.338,-178.434,5.954,148.597
C07299=1203.711,124.338,-51.358,-178.432,5.955,148.597
C07300=1203.706,124.587,-51.378,-178.429,5.956,148.596
C07301=1203.700,124.836,-51.397,-178.426,5.958,148.596
C07302=1203.696,125.085,-51.417,-178.424,5.959,148.595
C07303=1203.691,125.335,-51.437,-178.421,5.960,148.595
C07304=1203.686,125.584,-51.457,-178.419,5.961,148.594
C07305=1203.681,125.832,-51.477,-178.416,5.963,148.594
C07306=1203.677,126.082,-51.496,-178.414,5.963,148.593
C07307=1203.672,126.332,-51.516,-178.411,5.965,148.593
C07308=1203.668,126.580,-51.536,-178.408,5.966,148.592
C07309=1203.663,126.830,-51.556,-178.406,5.968,148.592
C07310=1203.658,127.078,-51.576,-178.402,5.969,148.591
C07311=1203.653,127.328,-51.596,-178.400,5.970,148.591
C07312=1203.648,127.577,-51.615,-178.398,5.972,148.591
C07313=1203.644,127.826,-51.636,-178.395,5.972,148.590
C07314=1203.638,128.075,-51.655,-178.392,5.974,148.590
C07315=1203.634,128.324,-51.675,-178.390,5.975,148.589
C07316=1203.629,128.574,-51.695,-178.387,5.977,148.588
C07317=1203.624,128.823,-51.716,-178.385,5.977,148.588
